LIN {X -0.059,Y -676.284,Z 1223.528,A 0.000,B 0.000,C 90.000,E1 131.024} C_DIS
LIN {X 0.179,Y -679.882,Z 1223.520,A 0.000,B 0.000,C 90.000,E1 129.564} C_DIS
LIN {X 0.002,Y -682.891,Z 1223.513,A 0.000,B 0.000,C 90.000,E1 128.382} C_DIS
LIN {X 0.032,Y -686.511,Z 1223.505,A 0.000,B 0.000,C 90.000,E1 126.950} C_DIS
LIN {X -0.093,Y -688.857,Z 1223.500,A 0.000,B 0.000,C 90.000,E1 126.011} C_DIS
LIN {X -0.354,Y -692.133,Z 1223.492,A 0.000,B 0.000,C 90.000,E1 124.612} C_DIS
LIN {X -0.210,Y -694.745,Z 1223.486,A 0.000,B 0.000,C 90.000,E1 123.420} C_DIS
LIN {X 0.177,Y -697.295,Z 1223.479,A 0.000,B 0.000,C 90.000,E1 122.212} C_DIS
LIN {X 0.274,Y -700.099,Z 1223.471,A 0.000,B 0.000,C 90.000,E1 120.797} C_DIS
LIN {X 0.130,Y -701.847,Z 1223.466,A 0.000,B 0.000,C 90.000,E1 119.873} C_DIS
LIN {X 0.287,Y -703.893,Z 1223.460,A 0.000,B 0.000,C 90.000,E1 118.693} C_DIS
LIN {X -0.100,Y -704.903,Z 1223.456,A 0.000,B 0.000,C 90.000,E1 118.025} C_DIS
LIN {X -0.188,Y -705.601,Z 1223.452,A 0.000,B 0.000,C 90.000,E1 117.334} C_DIS
LIN {X 0.351,Y -706.241,Z 1223.447,A 0.000,B 0.000,C 90.000,E1 116.360} C_DIS
LIN {X -0.348,Y -706.468,Z 1223.443,A 0.000,B 0.000,C 90.000,E1 115.720} C_DIS
LIN {X -0.408,Y -706.297,Z 1223.439,A 0.000,B 0.000,C 90.000,E1 115.027} C_DIS
LIN {X 0.176,Y -705.957,Z 1223.436,A 0.000,B 0.000,C 90.000,E1 114.515} C_DIS
LIN {X -0.177,Y -705.023,Z 1223.434,A 0.000,B 0.000,C 90.000,E1 114.079} C_DIS
LIN {X 0.110,Y -704.351,Z 1223.432,A 0.000,B 0.000,C 90.000,E1 113.823} C_DIS
LIN {X -0.251,Y -702.302,Z 1223.430,A 0.000,B 0.000,C 90.000,E1 113.387} C_DIS
LIN {X -0.112,Y -701.601,Z 1223.429,A 0.000,B 0.000,C 90.000,E1 113.259} C_DIS
LIN {X 0.025,Y -700.554,Z 1223.429,A 0.000,B 0.000,C 90.000,E1 113.131} C_DIS
LIN {X -0.062,Y -695.166,Z 1223.426,A 0.000,B 0.000,C 90.000,E1 112.695} C_DIS
LIN {X -0.096,Y -693.311,Z 1223.426,A 0.000,B 0.000,C 90.000,E1 112.589} C_DIS
LIN {X 0.260,Y -686.621,Z 1223.424,A 0.000,B 0.000,C 90.000,E1 112.333} C_DIS
LIN {X -0.232,Y -684.453,Z 1223.424,A 0.000,B 0.000,C 90.000,E1 112.333} C_DIS
LIN {X -0.007,Y -677.105,Z 1223.424,A 0.000,B 0.000,C 90.000,E1 112.280} C_DIS
LIN {X -0.061,Y -614.428,Z 1223.424,A 0.000,B 0.000,C 90.000,E1 112.280} C_DIS
LIN {X 0.085,Y -612.192,Z 1223.423,A 0.000,B 0.000,C 90.000,E1 112.153} C_DIS
LIN {X -0.235,Y -608.439,Z 1223.422,A 0.000,B 0.000,C 90.000,E1 111.897} C_DIS
LIN {X -0.060,Y -607.204,Z 1223.421,A 0.000,B 0.000,C 90.000,E1 111.770} C_DIS
LIN {X 0.199,Y -605.431,Z 1223.420,A 0.000,B 0.000,C 90.000,E1 111.535} C_DIS
LIN {X 0.044,Y -604.843,Z 1223.419,A 0.000,B 0.000,C 90.000,E1 111.354} C_DIS
LIN {X 0.323,Y -605.149,Z 1223.417,A 0.000,B 0.000,C 90.000,E1 111.099} C_DIS
LIN {X 0.288,Y -605.464,Z 1223.417,A 0.000,B 0.000,C 90.000,E1 110.972} C_DIS
LIN {X -0.099,Y -607.826,Z 1223.413,A 0.000,B 0.000,C 90.000,E1 110.355} C_DIS
LIN {X -0.270,Y -608.959,Z 1223.412,A 0.000,B 0.000,C 90.000,E1 110.120} C_DIS
LIN {X -0.091,Y -612.081,Z 1223.407,A 0.000,B 0.000,C 90.000,E1 109.322} C_DIS
LIN {X 0.203,Y -616.524,Z 1223.400,A 0.000,B 0.000,C 90.000,E1 108.000} C_DIS
LIN {X -0.038,Y -617.374,Z 1223.399,A 0.000,B 0.000,C 90.000,E1 107.764} C_DIS
LIN {X 0.266,Y -619.489,Z 1223.396,A 0.000,B 0.000,C 90.000,E1 107.221} C_DIS
LIN {X -0.074,Y -624.283,Z 1223.389,A 0.000,B 0.000,C 90.000,E1 105.969} C_DIS
LIN {X 0.274,Y -626.084,Z 1223.386,A 0.000,B 0.000,C 90.000,E1 105.426} C_DIS
LIN {X -0.339,Y -628.318,Z 1223.382,A 0.000,B 0.000,C 90.000,E1 104.717} C_DIS
LIN {X -0.168,Y -630.033,Z 1223.377,A 0.000,B 0.000,C 90.000,E1 103.939} C_DIS
LIN {X 0.057,Y -630.911,Z 1223.375,A 0.000,B 0.000,C 90.000,E1 103.411} C_DIS
LIN {X 0.290,Y -631.567,Z 1223.372,A 0.000,B 0.000,C 90.000,E1 102.883} C_DIS
LIN {X 0.339,Y -631.709,Z 1223.368,A 0.000,B 0.000,C 90.000,E1 102.119} C_DIS
LIN {X -0.167,Y -631.385,Z 1223.365,A 0.000,B 0.000,C 90.000,E1 101.658} C_DIS
LIN {X 0.072,Y -630.629,Z 1223.362,A 0.000,B 0.000,C 90.000,E1 101.130} C_DIS
LIN {X 0.108,Y -628.943,Z 1223.358,A 0.000,B 0.000,C 90.000,E1 100.366} C_DIS
LIN {X -0.202,Y -628.261,Z 1223.356,A 0.000,B 0.000,C 90.000,E1 100.141} C_DIS
LIN {X 0.216,Y -627.442,Z 1223.355,A 0.000,B 0.000,C 90.000,E1 99.849} C_DIS
LIN {X -0.195,Y -625.511,Z 1223.352,A 0.000,B 0.000,C 90.000,E1 99.378} C_DIS
LIN {X -0.104,Y -623.269,Z 1223.349,A 0.000,B 0.000,C 90.000,E1 98.859} C_DIS
LIN {X -0.026,Y -620.545,Z 1223.346,A 0.000,B 0.000,C 90.000,E1 98.341} C_DIS
LIN {X -0.256,Y -618.750,Z 1223.345,A 0.000,B 0.000,C 90.000,E1 98.106} C_DIS
LIN {X -0.207,Y -614.791,Z 1223.342,A 0.000,B 0.000,C 90.000,E1 97.587} C_DIS
LIN {X -0.016,Y -611.544,Z 1223.340,A 0.000,B 0.000,C 90.000,E1 97.182} C_DIS
LIN {X 0.019,Y -606.606,Z 1223.337,A 0.000,B 0.000,C 90.000,E1 96.663} C_DIS
LIN {X -0.266,Y -602.361,Z 1223.335,A 0.000,B 0.000,C 90.000,E1 96.315} C_DIS
LIN {X 0.299,Y -598.150,Z 1223.333,A 0.000,B 0.000,C 90.000,E1 95.910} C_DIS
LIN {X -0.153,Y -592.184,Z 1223.331,A 0.000,B 0.000,C 90.000,E1 95.511} C_DIS
LIN {X 0.039,Y -584.245,Z 1223.328,A 0.000,B 0.000,C 90.000,E1 94.992} C_DIS
LIN {X -0.114,Y -577.272,Z 1223.326,A 0.000,B 0.000,C 90.000,E1 94.645} C_DIS
LIN {X 0.264,Y -572.044,Z 1223.324,A 0.000,B 0.000,C 90.000,E1 94.359} C_DIS
LIN {X -0.023,Y -566.787,Z 1223.323,A 0.000,B 0.000,C 90.000,E1 94.073} C_DIS
LIN {X -0.250,Y -564.966,Z 1223.320,A 0.000,B 0.000,C 90.000,E1 93.669} C_DIS
LIN {X -0.066,Y -564.757,Z 1223.320,A 0.000,B 0.000,C 90.000,E1 93.612} C_DIS
LIN {X -0.108,Y -564.741,Z 1223.320,A 0.000,B 0.000,C 90.000,E1 93.612} C_DIS
LIN {X 0.082,Y -564.561,Z 1223.318,A 0.000,B 0.000,C 90.000,E1 93.154} C_DIS
LIN {X -0.022,Y -564.983,Z 1223.312,A 0.000,B 0.000,C 90.000,E1 92.064} C_DIS
LIN {X 0.216,Y -566.310,Z 1223.301,A 0.000,B 0.000,C 90.000,E1 90.115} C_DIS
LIN {X -0.215,Y -567.482,Z 1223.292,A 0.000,B 0.000,C 90.000,E1 88.511} C_DIS
LIN {X 0.105,Y -568.886,Z 1223.281,A 0.000,B 0.000,C 90.000,E1 86.560} C_DIS
LIN {X -0.225,Y -570.213,Z 1223.272,A 0.000,B 0.000,C 90.000,E1 84.951} C_DIS
LIN {X -0.091,Y -571.449,Z 1223.264,A 0.000,B 0.000,C 90.000,E1 83.571} C_DIS
LIN {X 0.124,Y -572.711,Z 1223.257,A 0.000,B 0.000,C 90.000,E1 82.186} C_DIS
LIN {X 0.079,Y -574.094,Z 1223.248,A 0.000,B 0.000,C 90.000,E1 80.557} C_DIS
LIN {X 0.227,Y -574.850,Z 1223.242,A 0.000,B 0.000,C 90.000,E1 79.454} C_DIS
LIN {X 0.223,Y -575.919,Z 1223.233,A 0.000,B 0.000,C 90.000,E1 77.825} C_DIS
LIN {X 0.273,Y -576.748,Z 1223.225,A 0.000,B 0.000,C 90.000,E1 76.464} C_DIS
LIN {X 0.001,Y -577.635,Z 1223.216,A 0.000,B 0.000,C 90.000,E1 74.866} C_DIS
LIN {X -0.262,Y -578.504,Z 1223.207,A 0.000,B 0.000,C 90.000,E1 73.268} C_DIS
LIN {X -0.178,Y -579.420,Z 1223.198,A 0.000,B 0.000,C 90.000,E1 71.638} C_DIS
LIN {X 0.281,Y -580.252,Z 1223.190,A 0.000,B 0.000,C 90.000,E1 70.242} C_DIS
LIN {X -0.044,Y -581.854,Z 1223.177,A 0.000,B 0.000,C 90.000,E1 67.847} C_DIS
LIN {X 0.121,Y -583.018,Z 1223.169,A 0.000,B 0.000,C 90.000,E1 66.485} C_DIS
LIN {X 0.007,Y -584.278,Z 1223.162,A 0.000,B 0.000,C 90.000,E1 65.153} C_DIS
LIN {X 0.205,Y -585.938,Z 1223.152,A 0.000,B 0.000,C 90.000,E1 63.256} C_DIS
LIN {X 0.173,Y -587.852,Z 1223.141,A 0.000,B 0.000,C 90.000,E1 61.385} C_DIS
LIN {X -0.115,Y -589.238,Z 1223.134,A 0.000,B 0.000,C 90.000,E1 60.078} C_DIS
LIN {X -0.087,Y -590.605,Z 1223.126,A 0.000,B 0.000,C 90.000,E1 58.742} C_DIS
LIN {X 0.281,Y -591.835,Z 1223.119,A 0.000,B 0.000,C 90.000,E1 57.375} C_DIS
LIN {X -0.149,Y -592.950,Z 1223.112,A 0.000,B 0.000,C 90.000,E1 56.087} C_DIS
LIN {X -0.235,Y -594.028,Z 1223.104,A 0.000,B 0.000,C 90.000,E1 54.769} C_DIS
LIN {X 0.043,Y -595.053,Z 1223.097,A 0.000,B 0.000,C 90.000,E1 53.417} C_DIS
LIN {X -0.134,Y -596.040,Z 1223.089,A 0.000,B 0.000,C 90.000,E1 52.110} C_DIS
LIN {X -0.295,Y -597.046,Z 1223.082,A 0.000,B 0.000,C 90.000,E1 50.803} C_DIS
LIN {X -0.065,Y -597.586,Z 1223.075,A 0.000,B 0.000,C 90.000,E1 49.461} C_DIS
LIN {X -0.281,Y -598.222,Z 1223.068,A 0.000,B 0.000,C 90.000,E1 48.162} C_DIS
LIN {X 0.352,Y -598.496,Z 1223.063,A 0.000,B 0.000,C 90.000,E1 47.310} C_DIS
LIN {X -0.076,Y -598.805,Z 1223.057,A 0.000,B 0.000,C 90.000,E1 46.296} C_DIS
LIN {X -0.085,Y -598.864,Z 1223.051,A 0.000,B 0.000,C 90.000,E1 45.243} C_DIS
LIN {X -0.092,Y -598.785,Z 1223.046,A 0.000,B 0.000,C 90.000,E1 44.190} C_DIS
LIN {X 0.109,Y -598.584,Z 1223.041,A 0.000,B 0.000,C 90.000,E1 43.380} C_DIS
LIN {X 0.122,Y -598.073,Z 1223.035,A 0.000,B 0.000,C 90.000,E1 42.324} C_DIS
LIN {X 0.310,Y -597.379,Z 1223.028,A 0.000,B 0.000,C 90.000,E1 40.987} C_DIS
LIN {X -0.301,Y -596.610,Z 1223.021,A 0.000,B 0.000,C 90.000,E1 39.725} C_DIS
LIN {X -0.086,Y -595.582,Z 1223.013,A 0.000,B 0.000,C 90.000,E1 38.382} C_DIS
LIN {X -0.015,Y -594.501,Z 1223.007,A 0.000,B 0.000,C 90.000,E1 37.317} C_DIS
LIN {X 0.048,Y -593.129,Z 1223.001,A 0.000,B 0.000,C 90.000,E1 36.251} C_DIS
LIN {X 0.091,Y -591.547,Z 1222.996,A 0.000,B 0.000,C 90.000,E1 35.185} C_DIS
LIN {X -0.100,Y -590.059,Z 1222.991,A 0.000,B 0.000,C 90.000,E1 34.405} C_DIS
LIN {X 0.177,Y -588.396,Z 1222.987,A 0.000,B 0.000,C 90.000,E1 33.579} C_DIS
LIN {X -0.247,Y -587.057,Z 1222.984,A 0.000,B 0.000,C 90.000,E1 33.086} C_DIS
LIN {X -0.138,Y -584.159,Z 1222.978,A 0.000,B 0.000,C 90.000,E1 32.005} C_DIS
LIN {X -0.098,Y -582.461,Z 1222.975,A 0.000,B 0.000,C 90.000,E1 31.465} C_DIS
LIN {X -0.071,Y -580.560,Z 1222.972,A 0.000,B 0.000,C 90.000,E1 30.924} C_DIS
LIN {X -0.204,Y -577.327,Z 1222.967,A 0.000,B 0.000,C 90.000,E1 30.129} C_DIS
LIN {X 0.284,Y -574.974,Z 1222.964,A 0.000,B 0.000,C 90.000,E1 29.539} C_DIS
LIN {X -0.027,Y -572.455,Z 1222.961,A 0.000,B 0.000,C 90.000,E1 29.027} C_DIS
LIN {X -0.164,Y -568.879,Z 1222.958,A 0.000,B 0.000,C 90.000,E1 28.359} C_DIS
LIN {X 0.072,Y -564.280,Z 1222.953,A 0.000,B 0.000,C 90.000,E1 27.513} C_DIS
LIN {X 0.099,Y -560.113,Z 1222.949,A 0.000,B 0.000,C 90.000,E1 26.821} C_DIS
LIN {X -0.161,Y -555.569,Z 1222.945,A 0.000,B 0.000,C 90.000,E1 26.155} C_DIS
LIN {X -0.095,Y -551.637,Z 1222.942,A 0.000,B 0.000,C 90.000,E1 25.591} C_DIS
LIN {X 0.063,Y -548.547,Z 1222.940,A 0.000,B 0.000,C 90.000,E1 25.155} C_DIS
LIN {X -0.168,Y -541.798,Z 1222.935,A 0.000,B 0.000,C 90.000,E1 24.335} C_DIS
LIN {X 0.024,Y -534.509,Z 1222.930,A 0.000,B 0.000,C 90.000,E1 23.462} C_DIS
LIN {X -0.138,Y -526.938,Z 1222.926,A 0.000,B 0.000,C 90.000,E1 22.642} C_DIS
LIN {X -0.090,Y -521.762,Z 1222.923,A 0.000,B 0.000,C 90.000,E1 22.078} C_DIS
LIN {X -0.152,Y -510.874,Z 1222.917,A 0.000,B 0.000,C 90.000,E1 20.972} C_DIS
LIN {X -0.057,Y -499.892,Z 1222.911,A 0.000,B 0.000,C 90.000,E1 19.885} C_DIS
LIN {X -0.074,Y -489.981,Z 1222.905,A 0.000,B 0.000,C 90.000,E1 18.960} C_DIS
LIN {X -0.159,Y -482.654,Z 1222.902,A 0.000,B 0.000,C 90.000,E1 18.308} C_DIS
LIN {X -0.043,Y -471.100,Z 1222.896,A 0.000,B 0.000,C 90.000,E1 17.275} C_DIS
LIN {X 0.101,Y -457.930,Z 1222.889,A 0.000,B 0.000,C 90.000,E1 16.079} C_DIS
LIN {X -0.247,Y -440.285,Z 1222.880,A 0.000,B 0.000,C 90.000,E1 14.481} C_DIS
LIN {X -0.047,Y -420.268,Z 1222.869,A 0.000,B 0.000,C 90.000,E1 12.411} C_DIS
LIN {X 0.106,Y -403.560,Z 1222.858,A 0.000,B 0.000,C 90.000,E1 10.489} C_DIS
LIN {X -0.208,Y -398.266,Z 1222.855,A 0.000,B 0.000,C 90.000,E1 9.849} C_DIS
LIN {X 0.192,Y -394.919,Z 1222.852,A 0.000,B 0.000,C 90.000,E1 9.265} C_DIS
LIN {X 0.114,Y -393.810,Z 1222.850,A 0.000,B 0.000,C 90.000,E1 8.973} C_DIS
LIN {X 0.076,Y -393.799,Z 1222.850,A 0.000,B 0.000,C 90.000,E1 8.973} C_DIS
LIN {X 0.084,Y -394.025,Z 1222.848,A 0.000,B 0.000,C 90.000,E1 8.690} C_DIS
LIN {X 0.105,Y -394.035,Z 1222.848,A 0.000,B 0.000,C 90.000,E1 8.681} C_DIS
LIN {X 0.042,Y -396.943,Z 1222.845,A 0.000,B 0.000,C 90.000,E1 8.049} C_DIS
LIN {X 0.063,Y -399.821,Z 1222.843,A 0.000,B 0.000,C 90.000,E1 7.701} C_DIS
LIN {X 0.073,Y -401.418,Z 1222.842,A 0.000,B 0.000,C 90.000,E1 7.530} C_DIS
LIN {X -0.127,Y -405.153,Z 1222.840,A 0.000,B 0.000,C 90.000,E1 7.239} C_DIS
LIN {X -0.195,Y -418.242,Z 1222.835,A 0.000,B 0.000,C 90.000,E1 6.258} C_DIS
LIN {X -0.178,Y -432.604,Z 1222.829,A 0.000,B 0.000,C 90.000,E1 5.163} C_DIS
LIN {X -0.107,Y -443.683,Z 1222.824,A 0.000,B 0.000,C 90.000,E1 4.302} C_DIS
LIN {X -0.046,Y -456.342,Z 1222.818,A 0.000,B 0.000,C 90.000,E1 3.326} C_DIS
LIN {X 0.101,Y -465.722,Z 1222.814,A 0.000,B 0.000,C 90.000,E1 2.579} C_DIS
LIN {X -0.192,Y -471.854,Z 1222.812,A 0.000,B 0.000,C 90.000,E1 2.121} C_DIS
LIN {X 0.171,Y -479.159,Z 1222.808,A 0.000,B 0.000,C 90.000,E1 1.432} C_DIS
LIN {X 0.000,Y -484.954,Z 1222.805,A 0.000,B 0.000,C 90.000,E1 0.917} C_DIS
LIN {X 0.212,Y -491.536,Z 1222.802,A 0.000,B 0.000,C 90.000,E1 0.229} C_DIS
LIN {X 0.170,Y -498.380,Z 1222.797,A 0.000,B 0.000,C 90.000,E1 359.484} C_DIS
LIN {X 0.158,Y -504.685,Z 1222.793,A 0.000,B 0.000,C 90.000,E1 358.740} C_DIS
LIN {X 0.201,Y -510.430,Z 1222.789,A 0.000,B 0.000,C 90.000,E1 357.993} C_DIS
LIN {X 0.243,Y -515.707,Z 1222.785,A 0.000,B 0.000,C 90.000,E1 357.249} C_DIS
LIN {X -0.163,Y -520.650,Z 1222.781,A 0.000,B 0.000,C 90.000,E1 356.560} C_DIS
LIN {X -0.277,Y -524.346,Z 1222.778,A 0.000,B 0.000,C 90.000,E1 355.988} C_DIS
LIN {X -0.087,Y -528.528,Z 1222.774,A 0.000,B 0.000,C 90.000,E1 355.241} C_DIS
LIN {X -0.108,Y -531.614,Z 1222.770,A 0.000,B 0.000,C 90.000,E1 354.666} C_DIS
LIN {X -0.068,Y -535.706,Z 1222.766,A 0.000,B 0.000,C 90.000,E1 353.799} C_DIS
LIN {X 0.239,Y -537.669,Z 1222.763,A 0.000,B 0.000,C 90.000,E1 353.337} C_DIS
LIN {X -0.185,Y -541.159,Z 1222.758,A 0.000,B 0.000,C 90.000,E1 352.527} C_DIS
LIN {X -0.117,Y -543.342,Z 1222.755,A 0.000,B 0.000,C 90.000,E1 351.951} C_DIS
LIN {X 0.050,Y -546.331,Z 1222.750,A 0.000,B 0.000,C 90.000,E1 351.084} C_DIS
LIN {X -0.296,Y -549.011,Z 1222.746,A 0.000,B 0.000,C 90.000,E1 350.274} C_DIS
LIN {X 0.251,Y -552.968,Z 1222.738,A 0.000,B 0.000,C 90.000,E1 348.814} C_DIS
LIN {X 0.202,Y -555.871,Z 1222.732,A 0.000,B 0.000,C 90.000,E1 347.701} C_DIS
LIN {X 0.056,Y -557.799,Z 1222.727,A 0.000,B 0.000,C 90.000,E1 346.881} C_DIS
LIN {X -0.197,Y -560.745,Z 1222.719,A 0.000,B 0.000,C 90.000,E1 345.519} C_DIS
LIN {X -0.005,Y -562.954,Z 1222.713,A 0.000,B 0.000,C 90.000,E1 344.393} C_DIS
LIN {X 0.212,Y -564.938,Z 1222.707,A 0.000,B 0.000,C 90.000,E1 343.268} C_DIS
LIN {X 0.078,Y -566.653,Z 1222.701,A 0.000,B 0.000,C 90.000,E1 342.181} C_DIS
LIN {X 0.309,Y -568.505,Z 1222.693,A 0.000,B 0.000,C 90.000,E1 340.786} C_DIS
LIN {X -0.119,Y -569.478,Z 1222.689,A 0.000,B 0.000,C 90.000,E1 340.007} C_DIS
LIN {X 0.186,Y -570.159,Z 1222.684,A 0.000,B 0.000,C 90.000,E1 339.156} C_DIS
LIN {X 0.175,Y -570.625,Z 1222.680,A 0.000,B 0.000,C 90.000,E1 338.337} C_DIS
LIN {X -0.038,Y -570.854,Z 1222.675,A 0.000,B 0.000,C 90.000,E1 337.539} C_DIS
LIN {X 0.097,Y -570.545,Z 1222.669,A 0.000,B 0.000,C 90.000,E1 336.433} C_DIS
LIN {X -0.247,Y -570.248,Z 1222.666,A 0.000,B 0.000,C 90.000,E1 335.921} C_DIS
LIN {X -0.242,Y -569.376,Z 1222.662,A 0.000,B 0.000,C 90.000,E1 335.101} C_DIS
LIN {X -0.246,Y -568.326,Z 1222.657,A 0.000,B 0.000,C 90.000,E1 334.280} C_DIS
LIN {X -0.013,Y -566.722,Z 1222.652,A 0.000,B 0.000,C 90.000,E1 333.435} C_DIS
LIN {X -0.049,Y -564.801,Z 1222.648,A 0.000,B 0.000,C 90.000,E1 332.615} C_DIS
LIN {X 0.340,Y -563.446,Z 1222.645,A 0.000,B 0.000,C 90.000,E1 332.025} C_DIS
LIN {X -0.042,Y -561.824,Z 1222.642,A 0.000,B 0.000,C 90.000,E1 331.513} C_DIS
LIN {X -0.238,Y -560.916,Z 1222.640,A 0.000,B 0.000,C 90.000,E1 331.257} C_DIS
LIN {X 0.123,Y -558.717,Z 1222.637,A 0.000,B 0.000,C 90.000,E1 330.667} C_DIS
LIN {X -0.234,Y -554.940,Z 1222.633,A 0.000,B 0.000,C 90.000,E1 329.871} C_DIS
LIN {X 0.126,Y -550.429,Z 1222.628,A 0.000,B 0.000,C 90.000,E1 328.997} C_DIS
LIN {X -0.193,Y -546.066,Z 1222.624,A 0.000,B 0.000,C 90.000,E1 328.329} C_DIS
LIN {X 0.200,Y -541.331,Z 1222.620,A 0.000,B 0.000,C 90.000,E1 327.582} C_DIS
LIN {X 0.082,Y -538.220,Z 1222.618,A 0.000,B 0.000,C 90.000,E1 327.168} C_DIS
LIN {X 0.233,Y -529.278,Z 1222.611,A 0.000,B 0.000,C 90.000,E1 326.008} C_DIS
LIN {X -0.133,Y -517.890,Z 1222.603,A 0.000,B 0.000,C 90.000,E1 324.609} C_DIS
LIN {X -0.023,Y -514.390,Z 1222.600,A 0.000,B 0.000,C 90.000,E1 324.069} C_DIS
LIN {X 0.074,Y -511.531,Z 1222.598,A 0.000,B 0.000,C 90.000,E1 323.543} C_DIS
LIN {X -0.008,Y -509.878,Z 1222.595,A 0.000,B 0.000,C 90.000,E1 323.084} C_DIS
LIN {X 0.103,Y -509.411,Z 1222.594,A 0.000,B 0.000,C 90.000,E1 322.924} C_DIS
LIN {X 0.088,Y -508.395,Z 1222.591,A 0.000,B 0.000,C 90.000,E1 322.396} C_DIS
LIN {X -0.004,Y -508.026,Z 1222.590,A 0.000,B 0.000,C 90.000,E1 322.110} C_DIS
LIN {X -0.159,Y -507.568,Z 1222.585,A 0.000,B 0.000,C 90.000,E1 321.251} C_DIS
LIN {X -0.036,Y -507.499,Z 1222.581,A 0.000,B 0.000,C 90.000,E1 320.642} C_DIS
LIN {X 0.049,Y -509.039,Z 1222.567,A 0.000,B 0.000,C 90.000,E1 317.957} C_DIS
LIN {X 0.188,Y -509.856,Z 1222.558,A 0.000,B 0.000,C 90.000,E1 316.458} C_DIS
LIN {X -0.021,Y -510.592,Z 1222.550,A 0.000,B 0.000,C 90.000,E1 315.000} C_DIS
LIN {X -0.066,Y -511.503,Z 1222.539,A 0.000,B 0.000,C 90.000,E1 312.933} C_DIS
LIN {X -0.057,Y -512.465,Z 1222.527,A 0.000,B 0.000,C 90.000,E1 310.862} C_DIS
LIN {X 0.193,Y -513.080,Z 1222.519,A 0.000,B 0.000,C 90.000,E1 309.358} C_DIS
LIN {X 0.280,Y -513.374,Z 1222.514,A 0.000,B 0.000,C 90.000,E1 308.463} C_DIS
LIN {X -0.015,Y -514.155,Z 1222.501,A 0.000,B 0.000,C 90.000,E1 306.137} C_DIS
LIN {X 0.087,Y -514.783,Z 1222.491,A 0.000,B 0.000,C 90.000,E1 304.358} C_DIS
LIN {X 0.144,Y -515.305,Z 1222.483,A 0.000,B 0.000,C 90.000,E1 302.880} C_DIS
LIN {X 0.081,Y -515.612,Z 1222.475,A 0.000,B 0.000,C 90.000,E1 301.416} C_DIS
LIN {X 0.033,Y -515.841,Z 1222.466,A 0.000,B 0.000,C 90.000,E1 299.951} C_DIS
LIN {X 0.075,Y -515.978,Z 1222.460,A 0.000,B 0.000,C 90.000,E1 298.771} C_DIS
LIN {X 0.015,Y -516.132,Z 1222.452,A 0.000,B 0.000,C 90.000,E1 297.308} C_DIS
LIN {X 0.060,Y -516.164,Z 1222.442,A 0.000,B 0.000,C 90.000,E1 295.540} C_DIS
LIN {X 0.117,Y -516.315,Z 1222.432,A 0.000,B 0.000,C 90.000,E1 293.770} C_DIS
LIN {X -0.169,Y -516.334,Z 1222.424,A 0.000,B 0.000,C 90.000,E1 292.333} C_DIS
LIN {X 0.011,Y -516.013,Z 1222.416,A 0.000,B 0.000,C 90.000,E1 290.844} C_DIS
LIN {X -0.133,Y -515.448,Z 1222.409,A 0.000,B 0.000,C 90.000,E1 289.685} C_DIS
LIN {X 0.280,Y -514.640,Z 1222.400,A 0.000,B 0.000,C 90.000,E1 287.873} C_DIS
LIN {X -0.083,Y -513.936,Z 1222.391,A 0.000,B 0.000,C 90.000,E1 286.441} C_DIS
LIN {X 0.039,Y -513.160,Z 1222.383,A 0.000,B 0.000,C 90.000,E1 284.954} C_DIS
LIN {X 0.075,Y -511.927,Z 1222.372,A 0.000,B 0.000,C 90.000,E1 282.883} C_DIS
LIN {X -0.082,Y -510.903,Z 1222.363,A 0.000,B 0.000,C 90.000,E1 281.422} C_DIS
LIN {X -0.183,Y -510.261,Z 1222.359,A 0.000,B 0.000,C 90.000,E1 280.546} C_DIS
LIN {X 0.005,Y -509.071,Z 1222.349,A 0.000,B 0.000,C 90.000,E1 278.746} C_DIS
LIN {X -0.008,Y -507.495,Z 1222.335,A 0.000,B 0.000,C 90.000,E1 276.372} C_DIS
LIN {X -0.194,Y -506.211,Z 1222.322,A 0.000,B 0.000,C 90.000,E1 274.012} C_DIS
LIN {X 0.020,Y -505.717,Z 1222.317,A 0.000,B 0.000,C 90.000,E1 273.094} C_DIS
LIN {X 0.010,Y -504.723,Z 1222.309,A 0.000,B 0.000,C 90.000,E1 271.604} C_DIS
LIN {X -0.024,Y -503.741,Z 1222.301,A 0.000,B 0.000,C 90.000,E1 270.115} C_DIS
LIN {X -0.076,Y -502.931,Z 1222.292,A 0.000,B 0.000,C 90.000,E1 268.625} C_DIS
LIN {X 0.155,Y -501.732,Z 1222.281,A 0.000,B 0.000,C 90.000,E1 266.502} C_DIS
LIN {X 0.194,Y -500.946,Z 1222.274,A 0.000,B 0.000,C 90.000,E1 265.298} C_DIS
LIN {X 0.175,Y -499.866,Z 1222.266,A 0.000,B 0.000,C 90.000,E1 263.799} C_DIS
LIN {X 0.222,Y -498.842,Z 1222.259,A 0.000,B 0.000,C 90.000,E1 262.591} C_DIS
LIN {X 0.060,Y -496.881,Z 1222.247,A 0.000,B 0.000,C 90.000,E1 260.500} C_DIS
LIN {X 0.030,Y -495.589,Z 1222.239,A 0.000,B 0.000,C 90.000,E1 258.993} C_DIS
LIN {X -0.105,Y -493.443,Z 1222.224,A 0.000,B 0.000,C 90.000,E1 256.284} C_DIS
LIN {X -0.010,Y -492.418,Z 1222.215,A 0.000,B 0.000,C 90.000,E1 254.755} C_DIS
LIN {X 0.173,Y -490.733,Z 1222.198,A 0.000,B 0.000,C 90.000,E1 251.692} C_DIS
LIN {X 0.036,Y -489.858,Z 1222.188,A 0.000,B 0.000,C 90.000,E1 249.880} C_DIS
LIN {X 0.156,Y -489.217,Z 1222.182,A 0.000,B 0.000,C 90.000,E1 248.646} C_DIS
LIN {X 0.269,Y -488.456,Z 1222.175,A 0.000,B 0.000,C 90.000,E1 247.411} C_DIS
LIN {X -0.081,Y -487.566,Z 1222.168,A 0.000,B 0.000,C 90.000,E1 246.230} C_DIS
LIN {X -0.218,Y -485.933,Z 1222.158,A 0.000,B 0.000,C 90.000,E1 244.409} C_DIS
LIN {X -0.191,Y -484.416,Z 1222.149,A 0.000,B 0.000,C 90.000,E1 242.871} C_DIS
LIN {X 0.246,Y -483.543,Z 1222.144,A 0.000,B 0.000,C 90.000,E1 241.897} C_DIS
LIN {X -0.188,Y -482.164,Z 1222.137,A 0.000,B 0.000,C 90.000,E1 240.717} C_DIS
LIN {X -0.197,Y -481.087,Z 1222.132,A 0.000,B 0.000,C 90.000,E1 239.793} C_DIS
LIN {X 0.195,Y -479.355,Z 1222.124,A 0.000,B 0.000,C 90.000,E1 238.201} C_DIS
LIN {X -0.073,Y -477.160,Z 1222.113,A 0.000,B 0.000,C 90.000,E1 236.373} C_DIS
LIN {X 0.106,Y -474.360,Z 1222.099,A 0.000,B 0.000,C 90.000,E1 233.863} C_DIS
LIN {X -0.006,Y -472.691,Z 1222.091,A 0.000,B 0.000,C 90.000,E1 232.316} C_DIS
LIN {X -0.139,Y -470.311,Z 1222.077,A 0.000,B 0.000,C 90.000,E1 229.828} C_DIS
LIN {X -0.016,Y -468.939,Z 1222.068,A 0.000,B 0.000,C 90.000,E1 228.243} C_DIS
LIN {X -0.130,Y -466.942,Z 1222.056,A 0.000,B 0.000,C 90.000,E1 226.053} C_DIS
LIN {X -0.138,Y -465.036,Z 1222.000,A 0.000,B 0.000,C 90.000,E1 215.931} C_DIS
LIN {X 0.059,Y -467.545,Z 1221.977,A 0.000,B 0.000,C 90.000,E1 211.799} C_DIS
LIN {X 0.198,Y -469.058,Z 1221.968,A 0.000,B 0.000,C 90.000,E1 210.207} C_DIS
LIN {X 0.169,Y -472.175,Z 1221.952,A 0.000,B 0.000,C 90.000,E1 207.385} C_DIS
LIN {X 0.050,Y -475.252,Z 1221.938,A 0.000,B 0.000,C 90.000,E1 204.899} C_DIS
LIN {X 0.043,Y -480.522,Z 1221.919,A 0.000,B 0.000,C 90.000,E1 201.482} C_DIS
LIN {X -0.233,Y -487.846,Z 1221.899,A 0.000,B 0.000,C 90.000,E1 197.819} C_DIS
LIN {X 0.130,Y -495.918,Z 1221.880,A 0.000,B 0.000,C 90.000,E1 194.426} C_DIS
LIN {X -0.225,Y -501.638,Z 1221.869,A 0.000,B 0.000,C 90.000,E1 192.355} C_DIS
LIN {X -0.057,Y -505.777,Z 1221.860,A 0.000,B 0.000,C 90.000,E1 190.838} C_DIS
LIN {X 0.029,Y -511.799,Z 1221.849,A 0.000,B 0.000,C 90.000,E1 188.746} C_DIS
LIN {X -0.203,Y -516.239,Z 1221.840,A 0.000,B 0.000,C 90.000,E1 187.296} C_DIS
LIN {X 0.106,Y -519.715,Z 1221.834,A 0.000,B 0.000,C 90.000,E1 186.087} C_DIS
LIN {X -0.160,Y -526.470,Z 1221.821,A 0.000,B 0.000,C 90.000,E1 183.784} C_DIS
LIN {X 0.246,Y -530.750,Z 1221.813,A 0.000,B 0.000,C 90.000,E1 182.293} C_DIS
LIN {X 0.203,Y -534.977,Z 1221.805,A 0.000,B 0.000,C 90.000,E1 180.859} C_DIS
LIN {X 0.226,Y -539.171,Z 1221.797,A 0.000,B 0.000,C 90.000,E1 179.427} C_DIS
LIN {X -0.179,Y -544.022,Z 1221.787,A 0.000,B 0.000,C 90.000,E1 177.764} C_DIS
LIN {X 0.018,Y -547.912,Z 1221.780,A 0.000,B 0.000,C 90.000,E1 176.331} C_DIS
LIN {X -0.230,Y -551.648,Z 1221.772,A 0.000,B 0.000,C 90.000,E1 174.951} C_DIS
LIN {X 0.134,Y -555.249,Z 1221.764,A 0.000,B 0.000,C 90.000,E1 173.514} C_DIS
LIN {X 0.067,Y -558.781,Z 1221.756,A 0.000,B 0.000,C 90.000,E1 172.129} C_DIS
LIN {X -0.005,Y -561.573,Z 1221.750,A 0.000,B 0.000,C 90.000,E1 171.027} C_DIS
LIN {X -0.038,Y -564.376,Z 1221.744,A 0.000,B 0.000,C 90.000,E1 169.926} C_DIS
LIN {X -0.136,Y -568.449,Z 1221.735,A 0.000,B 0.000,C 90.000,E1 168.285} C_DIS
LIN {X -0.142,Y -572.605,Z 1221.726,A 0.000,B 0.000,C 90.000,E1 166.645} C_DIS
LIN {X -0.284,Y -577.657,Z 1221.715,A 0.000,B 0.000,C 90.000,E1 164.755} C_DIS
LIN {X -0.039,Y -586.173,Z 1221.699,A 0.000,B 0.000,C 90.000,E1 161.764} C_DIS
LIN {X 0.065,Y -599.104,Z 1221.678,A 0.000,B 0.000,C 90.000,E1 158.028} C_DIS
LIN {X 0.072,Y -603.122,Z 1221.672,A 0.000,B 0.000,C 90.000,E1 156.975} C_DIS
LIN {X 0.130,Y -607.099,Z 1221.666,A 0.000,B 0.000,C 90.000,E1 155.921} C_DIS
LIN {X -0.363,Y -612.003,Z 1221.659,A 0.000,B 0.000,C 90.000,E1 154.665} C_DIS
LIN {X 0.059,Y -615.769,Z 1221.653,A 0.000,B 0.000,C 90.000,E1 153.589} C_DIS
LIN {X -0.020,Y -619.398,Z 1221.648,A 0.000,B 0.000,C 90.000,E1 152.564} C_DIS
LIN {X 0.239,Y -623.749,Z 1221.641,A 0.000,B 0.000,C 90.000,E1 151.257} C_DIS
LIN {X 0.022,Y -627.175,Z 1221.635,A 0.000,B 0.000,C 90.000,E1 150.255} C_DIS
LIN {X -0.124,Y -631.420,Z 1221.628,A 0.000,B 0.000,C 90.000,E1 148.997} C_DIS
LIN {X 0.158,Y -636.288,Z 1221.619,A 0.000,B 0.000,C 90.000,E1 147.454} C_DIS
LIN {X 0.064,Y -638.577,Z 1221.615,A 0.000,B 0.000,C 90.000,E1 146.707} C_DIS
LIN {X -0.105,Y -642.269,Z 1221.608,A 0.000,B 0.000,C 90.000,E1 145.468} C_DIS
LIN {X -0.330,Y -646.173,Z 1221.600,A 0.000,B 0.000,C 90.000,E1 143.989} C_DIS
LIN {X 0.038,Y -647.958,Z 1221.596,A 0.000,B 0.000,C 90.000,E1 143.210} C_DIS
LIN {X -0.203,Y -651.413,Z 1221.587,A 0.000,B 0.000,C 90.000,E1 141.743} C_DIS
LIN {X -0.318,Y -654.162,Z 1221.581,A 0.000,B 0.000,C 90.000,E1 140.517} C_DIS
LIN {X 0.018,Y -656.881,Z 1221.574,A 0.000,B 0.000,C 90.000,E1 139.256} C_DIS
LIN {X -0.132,Y -660.162,Z 1221.566,A 0.000,B 0.000,C 90.000,E1 137.796} C_DIS
LIN {X 0.222,Y -663.848,Z 1221.556,A 0.000,B 0.000,C 90.000,E1 136.053} C_DIS
LIN {X 0.200,Y -669.057,Z 1221.544,A 0.000,B 0.000,C 90.000,E1 133.866} C_DIS
LIN {X -0.211,Y -672.135,Z 1221.537,A 0.000,B 0.000,C 90.000,E1 132.690} C_DIS
LIN {X -0.052,Y -675.822,Z 1221.529,A 0.000,B 0.000,C 90.000,E1 131.229} C_DIS
LIN {X -0.237,Y -679.972,Z 1221.520,A 0.000,B 0.000,C 90.000,E1 129.564} C_DIS
LIN {X 0.122,Y -682.964,Z 1221.513,A 0.000,B 0.000,C 90.000,E1 128.338} C_DIS
LIN {X -0.384,Y -686.599,Z 1221.505,A 0.000,B 0.000,C 90.000,E1 126.950} C_DIS
LIN {X 0.049,Y -688.934,Z 1221.500,A 0.000,B 0.000,C 90.000,E1 125.964} C_DIS
LIN {X 0.190,Y -692.230,Z 1221.492,A 0.000,B 0.000,C 90.000,E1 124.532} C_DIS
LIN {X -0.398,Y -695.339,Z 1221.484,A 0.000,B 0.000,C 90.000,E1 123.166} C_DIS
LIN {X -0.241,Y -697.365,Z 1221.479,A 0.000,B 0.000,C 90.000,E1 122.212} C_DIS
LIN {X -0.144,Y -700.193,Z 1221.471,A 0.000,B 0.000,C 90.000,E1 120.797} C_DIS
LIN {X -0.352,Y -702.788,Z 1221.463,A 0.000,B 0.000,C 90.000,E1 119.411} C_DIS
LIN {X 0.153,Y -704.332,Z 1221.458,A 0.000,B 0.000,C 90.000,E1 118.437} C_DIS
LIN {X -0.232,Y -705.232,Z 1221.454,A 0.000,B 0.000,C 90.000,E1 117.769} C_DIS
LIN {X 0.007,Y -705.859,Z 1221.450,A 0.000,B 0.000,C 90.000,E1 117.052} C_DIS
LIN {X 0.228,Y -706.403,Z 1221.445,A 0.000,B 0.000,C 90.000,E1 116.104} C_DIS
LIN {X 0.168,Y -706.499,Z 1221.441,A 0.000,B 0.000,C 90.000,E1 115.412} C_DIS
LIN {X 0.115,Y -706.355,Z 1221.439,A 0.000,B 0.000,C 90.000,E1 114.951} C_DIS
LIN {X -0.238,Y -705.958,Z 1221.436,A 0.000,B 0.000,C 90.000,E1 114.515} C_DIS
LIN {X 0.052,Y -705.000,Z 1221.434,A 0.000,B 0.000,C 90.000,E1 114.027} C_DIS
LIN {X -0.303,Y -704.241,Z 1221.432,A 0.000,B 0.000,C 90.000,E1 113.823} C_DIS
LIN {X -0.019,Y -702.197,Z 1221.430,A 0.000,B 0.000,C 90.000,E1 113.334} C_DIS
LIN {X 0.120,Y -701.412,Z 1221.429,A 0.000,B 0.000,C 90.000,E1 113.206} C_DIS
LIN {X 0.258,Y -700.245,Z 1221.428,A 0.000,B 0.000,C 90.000,E1 113.078} C_DIS
LIN {X 0.170,Y -694.653,Z 1221.426,A 0.000,B 0.000,C 90.000,E1 112.642} C_DIS
LIN {X -0.175,Y -692.571,Z 1221.425,A 0.000,B 0.000,C 90.000,E1 112.567} C_DIS
LIN {X 0.023,Y -685.847,Z 1221.424,A 0.000,B 0.000,C 90.000,E1 112.333} C_DIS
LIN {X -0.226,Y -684.511,Z 1221.424,A 0.000,B 0.000,C 90.000,E1 112.333} C_DIS
LIN {X 0.014,Y -676.884,Z 1221.424,A 0.000,B 0.000,C 90.000,E1 112.280} C_DIS
LIN {X -0.020,Y -613.742,Z 1221.424,A 0.000,B 0.000,C 90.000,E1 112.280} C_DIS
LIN {X -0.024,Y -611.226,Z 1221.423,A 0.000,B 0.000,C 90.000,E1 112.153} C_DIS
LIN {X 0.033,Y -607.187,Z 1221.421,A 0.000,B 0.000,C 90.000,E1 111.844} C_DIS
LIN {X -0.061,Y -605.331,Z 1221.420,A 0.000,B 0.000,C 90.000,E1 111.642} C_DIS
LIN {X 0.119,Y -603.890,Z 1221.419,A 0.000,B 0.000,C 90.000,E1 111.482} C_DIS
LIN {X 0.076,Y -603.851,Z 1221.419,A 0.000,B 0.000,C 90.000,E1 111.482} C_DIS
LIN {X 0.308,Y -603.272,Z 1221.418,A 0.000,B 0.000,C 90.000,E1 111.280} C_DIS
LIN {X 0.070,Y -604.117,Z 1221.416,A 0.000,B 0.000,C 90.000,E1 110.844} C_DIS
LIN {X -0.180,Y -605.884,Z 1221.413,A 0.000,B 0.000,C 90.000,E1 110.355} C_DIS
LIN {X -0.239,Y -609.035,Z 1221.409,A 0.000,B 0.000,C 90.000,E1 109.577} C_DIS
LIN {X -0.320,Y -612.624,Z 1221.403,A 0.000,B 0.000,C 90.000,E1 108.544} C_DIS
LIN {X -0.299,Y -615.175,Z 1221.399,A 0.000,B 0.000,C 90.000,E1 107.764} C_DIS
LIN {X -0.011,Y -617.121,Z 1221.396,A 0.000,B 0.000,C 90.000,E1 107.221} C_DIS
LIN {X -0.170,Y -620.941,Z 1221.390,A 0.000,B 0.000,C 90.000,E1 106.205} C_DIS
LIN {X -0.064,Y -623.478,Z 1221.386,A 0.000,B 0.000,C 90.000,E1 105.426} C_DIS
LIN {X -0.097,Y -625.555,Z 1221.381,A 0.000,B 0.000,C 90.000,E1 104.662} C_DIS
LIN {X 0.253,Y -626.750,Z 1221.379,A 0.000,B 0.000,C 90.000,E1 104.120} C_DIS
LIN {X -0.154,Y -627.648,Z 1221.376,A 0.000,B 0.000,C 90.000,E1 103.647} C_DIS
LIN {X 0.056,Y -628.291,Z 1221.373,A 0.000,B 0.000,C 90.000,E1 103.119} C_DIS
LIN {X -0.143,Y -628.508,Z 1221.372,A 0.000,B 0.000,C 90.000,E1 102.883} C_DIS
LIN {X 0.074,Y -628.661,Z 1221.369,A 0.000,B 0.000,C 90.000,E1 102.355} C_DIS
LIN {X 0.292,Y -628.375,Z 1221.366,A 0.000,B 0.000,C 90.000,E1 101.827} C_DIS
LIN {X 0.093,Y -628.085,Z 1221.365,A 0.000,B 0.000,C 90.000,E1 101.591} C_DIS
LIN {X 0.185,Y -627.210,Z 1221.362,A 0.000,B 0.000,C 90.000,E1 101.074} C_DIS
LIN {X -0.221,Y -626.120,Z 1221.359,A 0.000,B 0.000,C 90.000,E1 100.602} C_DIS
LIN {X -0.023,Y -624.646,Z 1221.356,A 0.000,B 0.000,C 90.000,E1 100.074} C_DIS
LIN {X 0.057,Y -622.752,Z 1221.353,A 0.000,B 0.000,C 90.000,E1 99.557} C_DIS
LIN {X 0.067,Y -619.904,Z 1221.350,A 0.000,B 0.000,C 90.000,E1 98.916} C_DIS
LIN {X 0.044,Y -616.126,Z 1221.346,A 0.000,B 0.000,C 90.000,E1 98.276} C_DIS
LIN {X 0.070,Y -612.332,Z 1221.343,A 0.000,B 0.000,C 90.000,E1 97.757} C_DIS
LIN {X -0.102,Y -606.514,Z 1221.340,A 0.000,B 0.000,C 90.000,E1 97.125} C_DIS
LIN {X 0.023,Y -601.218,Z 1221.337,A 0.000,B 0.000,C 90.000,E1 96.606} C_DIS
LIN {X -0.112,Y -595.675,Z 1221.334,A 0.000,B 0.000,C 90.000,E1 96.144} C_DIS
LIN {X 0.104,Y -589.615,Z 1221.332,A 0.000,B 0.000,C 90.000,E1 95.682} C_DIS
LIN {X 0.267,Y -586.410,Z 1221.330,A 0.000,B 0.000,C 90.000,E1 95.454} C_DIS
LIN {X 0.075,Y -578.178,Z 1221.328,A 0.000,B 0.000,C 90.000,E1 94.992} C_DIS
LIN {X 0.153,Y -571.237,Z 1221.326,A 0.000,B 0.000,C 90.000,E1 94.645} C_DIS
LIN {X -0.051,Y -567.372,Z 1221.325,A 0.000,B 0.000,C 90.000,E1 94.416} C_DIS
LIN {X -0.173,Y -564.449,Z 1221.322,A 0.000,B 0.000,C 90.000,E1 94.012} C_DIS
LIN {X 0.048,Y -564.342,Z 1221.321,A 0.000,B 0.000,C 90.000,E1 93.784} C_DIS
LIN {X -0.066,Y -564.543,Z 1221.315,A 0.000,B 0.000,C 90.000,E1 92.694} C_DIS
LIN {X 0.269,Y -565.993,Z 1221.303,A 0.000,B 0.000,C 90.000,E1 90.458} C_DIS
LIN {X -0.166,Y -567.166,Z 1221.294,A 0.000,B 0.000,C 90.000,E1 88.854} C_DIS
LIN {X 0.118,Y -568.570,Z 1221.283,A 0.000,B 0.000,C 90.000,E1 86.906} C_DIS
LIN {X -0.229,Y -569.878,Z 1221.274,A 0.000,B 0.000,C 90.000,E1 85.298} C_DIS
LIN {X 0.073,Y -571.310,Z 1221.265,A 0.000,B 0.000,C 90.000,E1 83.628} C_DIS
LIN {X -0.089,Y -572.774,Z 1221.256,A 0.000,B 0.000,C 90.000,E1 82.008} C_DIS
LIN {X -0.219,Y -574.140,Z 1221.247,A 0.000,B 0.000,C 90.000,E1 80.387} C_DIS
LIN {X -0.078,Y -574.863,Z 1221.240,A 0.000,B 0.000,C 90.000,E1 79.285} C_DIS
LIN {X -0.178,Y -575.717,Z 1221.233,A 0.000,B 0.000,C 90.000,E1 77.937} C_DIS
LIN {X 0.092,Y -576.385,Z 1221.227,A 0.000,B 0.000,C 90.000,E1 76.825} C_DIS
LIN {X 0.155,Y -577.125,Z 1221.219,A 0.000,B 0.000,C 90.000,E1 75.463} C_DIS
LIN {X 0.231,Y -577.858,Z 1221.212,A 0.000,B 0.000,C 90.000,E1 74.102} C_DIS
LIN {X -0.047,Y -578.894,Z 1221.201,A 0.000,B 0.000,C 90.000,E1 72.236} C_DIS
LIN {X 0.185,Y -579.373,Z 1221.197,A 0.000,B 0.000,C 90.000,E1 71.402} C_DIS
LIN {X 0.092,Y -580.182,Z 1221.189,A 0.000,B 0.000,C 90.000,E1 70.061} C_DIS
LIN {X -0.096,Y -581.656,Z 1221.177,A 0.000,B 0.000,C 90.000,E1 67.922} C_DIS
LIN {X -0.077,Y -583.020,Z 1221.168,A 0.000,B 0.000,C 90.000,E1 66.305} C_DIS
LIN {X -0.068,Y -584.083,Z 1221.162,A 0.000,B 0.000,C 90.000,E1 65.229} C_DIS
LIN {X 0.117,Y -585.745,Z 1221.152,A 0.000,B 0.000,C 90.000,E1 63.332} C_DIS
LIN {X 0.238,Y -587.920,Z 1221.140,A 0.000,B 0.000,C 90.000,E1 61.179} C_DIS
LIN {X -0.046,Y -589.311,Z 1221.133,A 0.000,B 0.000,C 90.000,E1 59.871} C_DIS
LIN {X 0.101,Y -590.389,Z 1221.127,A 0.000,B 0.000,C 90.000,E1 58.791} C_DIS
LIN {X 0.153,Y -591.624,Z 1221.119,A 0.000,B 0.000,C 90.000,E1 57.454} C_DIS
LIN {X 0.047,Y -592.724,Z 1221.112,A 0.000,B 0.000,C 90.000,E1 56.135} C_DIS
LIN {X -0.034,Y -593.830,Z 1221.105,A 0.000,B 0.000,C 90.000,E1 54.815} C_DIS
LIN {X -0.136,Y -595.249,Z 1221.094,A 0.000,B 0.000,C 90.000,E1 52.970} C_DIS
LIN {X 0.154,Y -596.607,Z 1221.084,A 0.000,B 0.000,C 90.000,E1 51.090} C_DIS
LIN {X -0.002,Y -597.075,Z 1221.080,A 0.000,B 0.000,C 90.000,E1 50.312} C_DIS
LIN {X 0.390,Y -597.998,Z 1221.068,A 0.000,B 0.000,C 90.000,E1 48.162} C_DIS
LIN {X 0.175,Y -598.276,Z 1221.063,A 0.000,B 0.000,C 90.000,E1 47.391} C_DIS
LIN {X 0.374,Y -598.658,Z 1221.056,A 0.000,B 0.000,C 90.000,E1 46.053} C_DIS
LIN {X -0.059,Y -598.693,Z 1221.050,A 0.000,B 0.000,C 90.000,E1 45.040} C_DIS
LIN {X 0.354,Y -598.543,Z 1221.044,A 0.000,B 0.000,C 90.000,E1 43.947} C_DIS
LIN {X 0.142,Y -598.300,Z 1221.040,A 0.000,B 0.000,C 90.000,E1 43.176} C_DIS
LIN {X 0.118,Y -597.469,Z 1221.031,A 0.000,B 0.000,C 90.000,E1 41.595} C_DIS
LIN {X 0.120,Y -597.236,Z 1221.028,A 0.000,B 0.000,C 90.000,E1 41.067} C_DIS
LIN {X -0.111,Y -596.403,Z 1221.021,A 0.000,B 0.000,C 90.000,E1 39.769} C_DIS
LIN {X -0.279,Y -595.383,Z 1221.014,A 0.000,B 0.000,C 90.000,E1 38.463} C_DIS
LIN {X -0.071,Y -594.626,Z 1221.009,A 0.000,B 0.000,C 90.000,E1 37.649} C_DIS
LIN {X -0.014,Y -593.297,Z 1221.003,A 0.000,B 0.000,C 90.000,E1 36.583} C_DIS
LIN {X -0.187,Y -592.187,Z 1220.999,A 0.000,B 0.000,C 90.000,E1 35.804} C_DIS
LIN {X -0.165,Y -590.462,Z 1220.993,A 0.000,B 0.000,C 90.000,E1 34.739} C_DIS
LIN {X -0.013,Y -588.265,Z 1220.987,A 0.000,B 0.000,C 90.000,E1 33.658} C_DIS
LIN {X 0.185,Y -587.686,Z 1220.986,A 0.000,B 0.000,C 90.000,E1 33.372} C_DIS
LIN {X -0.192,Y -584.722,Z 1220.980,A 0.000,B 0.000,C 90.000,E1 32.339} C_DIS
LIN {X -0.284,Y -582.354,Z 1220.975,A 0.000,B 0.000,C 90.000,E1 31.544} C_DIS
LIN {X -0.098,Y -579.374,Z 1220.971,A 0.000,B 0.000,C 90.000,E1 30.718} C_DIS
LIN {X 0.255,Y -576.081,Z 1220.966,A 0.000,B 0.000,C 90.000,E1 29.873} C_DIS
LIN {X 0.074,Y -572.320,Z 1220.962,A 0.000,B 0.000,C 90.000,E1 29.077} C_DIS
LIN {X -0.068,Y -568.798,Z 1220.958,A 0.000,B 0.000,C 90.000,E1 28.409} C_DIS
LIN {X 0.082,Y -565.764,Z 1220.955,A 0.000,B 0.000,C 90.000,E1 27.847} C_DIS
LIN {X -0.027,Y -562.542,Z 1220.952,A 0.000,B 0.000,C 90.000,E1 27.308} C_DIS
LIN {X 0.084,Y -559.126,Z 1220.949,A 0.000,B 0.000,C 90.000,E1 26.744} C_DIS
LIN {X 0.174,Y -555.494,Z 1220.946,A 0.000,B 0.000,C 90.000,E1 26.181} C_DIS
LIN {X -0.017,Y -551.600,Z 1220.943,A 0.000,B 0.000,C 90.000,E1 25.643} C_DIS
LIN {X 0.019,Y -547.391,Z 1220.939,A 0.000,B 0.000,C 90.000,E1 25.079} C_DIS
LIN {X -0.098,Y -541.777,Z 1220.935,A 0.000,B 0.000,C 90.000,E1 24.387} C_DIS
LIN {X 0.227,Y -535.768,Z 1220.932,A 0.000,B 0.000,C 90.000,E1 23.643} C_DIS
LIN {X -0.009,Y -527.000,Z 1220.926,A 0.000,B 0.000,C 90.000,E1 22.695} C_DIS
LIN {X 0.184,Y -520.436,Z 1220.922,A 0.000,B 0.000,C 90.000,E1 21.972} C_DIS
LIN {X -0.196,Y -511.034,Z 1220.917,A 0.000,B 0.000,C 90.000,E1 21.046} C_DIS
LIN {X -0.021,Y -499.944,Z 1220.911,A 0.000,B 0.000,C 90.000,E1 19.939} C_DIS
LIN {X -0.233,Y -489.939,Z 1220.906,A 0.000,B 0.000,C 90.000,E1 19.033} C_DIS
LIN {X -0.154,Y -482.675,Z 1220.902,A 0.000,B 0.000,C 90.000,E1 18.362} C_DIS
LIN {X 0.039,Y -474.092,Z 1220.898,A 0.000,B 0.000,C 90.000,E1 17.583} C_DIS
LIN {X -0.224,Y -458.289,Z 1220.890,A 0.000,B 0.000,C 90.000,E1 16.205} C_DIS
LIN {X -0.024,Y -440.599,Z 1220.881,A 0.000,B 0.000,C 90.000,E1 14.537} C_DIS
LIN {X 0.100,Y -420.582,Z 1220.870,A 0.000,B 0.000,C 90.000,E1 12.479} C_DIS
LIN {X 0.076,Y -402.713,Z 1220.858,A 0.000,B 0.000,C 90.000,E1 10.433} C_DIS
LIN {X 0.066,Y -397.834,Z 1220.854,A 0.000,B 0.000,C 90.000,E1 9.792} C_DIS
LIN {X 0.166,Y -394.614,Z 1220.852,A 0.000,B 0.000,C 90.000,E1 9.265} C_DIS
LIN {X 0.135,Y -393.654,Z 1220.850,A 0.000,B 0.000,C 90.000,E1 8.973} C_DIS
LIN {X 0.097,Y -393.647,Z 1220.850,A 0.000,B 0.000,C 90.000,E1 8.973} C_DIS
LIN {X 0.020,Y -393.848,Z 1220.849,A 0.000,B 0.000,C 90.000,E1 8.746} C_DIS
LIN {X -0.018,Y -393.870,Z 1220.849,A 0.000,B 0.000,C 90.000,E1 8.746} C_DIS
LIN {X -0.188,Y -396.547,Z 1220.845,A 0.000,B 0.000,C 90.000,E1 8.163} C_DIS
LIN {X -0.014,Y -397.064,Z 1220.845,A 0.000,B 0.000,C 90.000,E1 8.049} C_DIS
LIN {X -0.176,Y -400.641,Z 1220.842,A 0.000,B 0.000,C 90.000,E1 7.644} C_DIS
LIN {X 0.173,Y -405.888,Z 1220.840,A 0.000,B 0.000,C 90.000,E1 7.125} C_DIS
LIN {X -0.134,Y -420.076,Z 1220.834,A 0.000,B 0.000,C 90.000,E1 6.087} C_DIS
LIN {X -0.008,Y -431.257,Z 1220.829,A 0.000,B 0.000,C 90.000,E1 5.220} C_DIS
LIN {X 0.019,Y -443.944,Z 1220.824,A 0.000,B 0.000,C 90.000,E1 4.245} C_DIS
LIN {X 0.122,Y -456.605,Z 1220.818,A 0.000,B 0.000,C 90.000,E1 3.269} C_DIS
LIN {X -0.179,Y -465.957,Z 1220.814,A 0.000,B 0.000,C 90.000,E1 2.579} C_DIS
LIN {X 0.025,Y -472.084,Z 1220.812,A 0.000,B 0.000,C 90.000,E1 2.064} C_DIS
LIN {X -0.061,Y -479.405,Z 1220.808,A 0.000,B 0.000,C 90.000,E1 1.432} C_DIS
LIN {X -0.214,Y -485.199,Z 1220.805,A 0.000,B 0.000,C 90.000,E1 0.917} C_DIS
LIN {X -0.195,Y -492.045,Z 1220.801,A 0.000,B 0.000,C 90.000,E1 0.229} C_DIS
LIN {X 0.170,Y -498.487,Z 1220.797,A 0.000,B 0.000,C 90.000,E1 359.484} C_DIS
LIN {X 0.232,Y -504.769,Z 1220.793,A 0.000,B 0.000,C 90.000,E1 358.740} C_DIS
LIN {X -0.198,Y -510.535,Z 1220.789,A 0.000,B 0.000,C 90.000,E1 358.051} C_DIS
LIN {X -0.158,Y -515.859,Z 1220.785,A 0.000,B 0.000,C 90.000,E1 357.306} C_DIS
LIN {X -0.047,Y -520.828,Z 1220.781,A 0.000,B 0.000,C 90.000,E1 356.560} C_DIS
LIN {X -0.159,Y -524.542,Z 1220.778,A 0.000,B 0.000,C 90.000,E1 355.988} C_DIS
LIN {X 0.034,Y -528.755,Z 1220.774,A 0.000,B 0.000,C 90.000,E1 355.241} C_DIS
LIN {X 0.016,Y -531.854,Z 1220.770,A 0.000,B 0.000,C 90.000,E1 354.666} C_DIS
LIN {X 0.059,Y -535.970,Z 1220.766,A 0.000,B 0.000,C 90.000,E1 353.799} C_DIS
LIN {X -0.168,Y -537.940,Z 1220.763,A 0.000,B 0.000,C 90.000,E1 353.394} C_DIS
LIN {X -0.053,Y -541.431,Z 1220.759,A 0.000,B 0.000,C 90.000,E1 352.527} C_DIS
LIN {X 0.018,Y -543.649,Z 1220.755,A 0.000,B 0.000,C 90.000,E1 351.951} C_DIS
LIN {X 0.189,Y -546.608,Z 1220.751,A 0.000,B 0.000,C 90.000,E1 351.084} C_DIS
LIN {X -0.153,Y -549.322,Z 1220.746,A 0.000,B 0.000,C 90.000,E1 350.274} C_DIS
LIN {X -0.142,Y -553.282,Z 1220.738,A 0.000,B 0.000,C 90.000,E1 348.870} C_DIS
LIN {X -0.186,Y -556.185,Z 1220.732,A 0.000,B 0.000,C 90.000,E1 347.757} C_DIS
LIN {X -0.191,Y -558.753,Z 1220.726,A 0.000,B 0.000,C 90.000,E1 346.645} C_DIS
LIN {X 0.115,Y -561.674,Z 1220.718,A 0.000,B 0.000,C 90.000,E1 345.227} C_DIS
LIN {X 0.166,Y -563.302,Z 1220.713,A 0.000,B 0.000,C 90.000,E1 344.393} C_DIS
LIN {X -0.152,Y -565.320,Z 1220.707,A 0.000,B 0.000,C 90.000,E1 343.323} C_DIS
LIN {X 0.261,Y -567.062,Z 1220.701,A 0.000,B 0.000,C 90.000,E1 342.181} C_DIS
LIN {X -0.224,Y -568.975,Z 1220.694,A 0.000,B 0.000,C 90.000,E1 340.859} C_DIS
LIN {X 0.077,Y -569.962,Z 1220.689,A 0.000,B 0.000,C 90.000,E1 340.007} C_DIS
LIN {X -0.146,Y -570.702,Z 1220.684,A 0.000,B 0.000,C 90.000,E1 339.209} C_DIS
LIN {X 0.171,Y -571.203,Z 1220.680,A 0.000,B 0.000,C 90.000,E1 338.358} C_DIS
LIN {X 0.004,Y -571.446,Z 1220.674,A 0.000,B 0.000,C 90.000,E1 337.283} C_DIS
LIN {X 0.148,Y -571.130,Z 1220.668,A 0.000,B 0.000,C 90.000,E1 336.177} C_DIS
LIN {X 0.161,Y -570.459,Z 1220.663,A 0.000,B 0.000,C 90.000,E1 335.357} C_DIS
LIN {X -0.005,Y -569.113,Z 1220.657,A 0.000,B 0.000,C 90.000,E1 334.280} C_DIS
LIN {X 0.159,Y -568.153,Z 1220.654,A 0.000,B 0.000,C 90.000,E1 333.717} C_DIS
LIN {X -0.115,Y -566.424,Z 1220.650,A 0.000,B 0.000,C 90.000,E1 332.922} C_DIS
LIN {X -0.158,Y -564.380,Z 1220.645,A 0.000,B 0.000,C 90.000,E1 332.103} C_DIS
LIN {X 0.227,Y -562.850,Z 1220.642,A 0.000,B 0.000,C 90.000,E1 331.513} C_DIS
LIN {X 0.112,Y -560.912,Z 1220.639,A 0.000,B 0.000,C 90.000,E1 330.973} C_DIS
LIN {X -0.287,Y -558.666,Z 1220.636,A 0.000,B 0.000,C 90.000,E1 330.461} C_DIS
LIN {X 0.162,Y -556.759,Z 1220.633,A 0.000,B 0.000,C 90.000,E1 329.999} C_DIS
LIN {X 0.009,Y -553.929,Z 1220.630,A 0.000,B 0.000,C 90.000,E1 329.459} C_DIS
LIN {X 0.193,Y -550.022,Z 1220.626,A 0.000,B 0.000,C 90.000,E1 328.742} C_DIS
LIN {X 0.029,Y -544.569,Z 1220.622,A 0.000,B 0.000,C 90.000,E1 327.916} C_DIS
LIN {X -0.072,Y -541.677,Z 1220.620,A 0.000,B 0.000,C 90.000,E1 327.502} C_DIS
LIN {X -0.013,Y -536.208,Z 1220.615,A 0.000,B 0.000,C 90.000,E1 326.786} C_DIS
LIN {X -0.178,Y -528.327,Z 1220.610,A 0.000,B 0.000,C 90.000,E1 325.801} C_DIS
LIN {X -0.050,Y -518.006,Z 1220.603,A 0.000,B 0.000,C 90.000,E1 324.482} C_DIS
LIN {X -0.301,Y -514.534,Z 1220.600,A 0.000,B 0.000,C 90.000,E1 323.989} C_DIS
LIN {X 0.269,Y -511.680,Z 1220.597,A 0.000,B 0.000,C 90.000,E1 323.417} C_DIS
LIN {X -0.056,Y -509.598,Z 1220.594,A 0.000,B 0.000,C 90.000,E1 322.844} C_DIS
LIN {X -0.032,Y -508.733,Z 1220.591,A 0.000,B 0.000,C 90.000,E1 322.396} C_DIS
LIN {X -0.122,Y -508.341,Z 1220.589,A 0.000,B 0.000,C 90.000,E1 322.110} C_DIS
LIN {X -0.308,Y -507.952,Z 1220.586,A 0.000,B 0.000,C 90.000,E1 321.537} C_DIS
LIN {X 0.114,Y -507.827,Z 1220.581,A 0.000,B 0.000,C 90.000,E1 320.598} C_DIS
LIN {X 0.157,Y -509.339,Z 1220.566,A 0.000,B 0.000,C 90.000,E1 317.919} C_DIS
LIN {X -0.041,Y -510.171,Z 1220.558,A 0.000,B 0.000,C 90.000,E1 316.458} C_DIS
LIN {X -0.244,Y -510.926,Z 1220.550,A 0.000,B 0.000,C 90.000,E1 315.000} C_DIS
LIN {X -0.183,Y -511.713,Z 1220.540,A 0.000,B 0.000,C 90.000,E1 313.218} C_DIS
LIN {X -0.089,Y -512.564,Z 1220.530,A 0.000,B 0.000,C 90.000,E1 311.434} C_DIS
LIN {X 0.155,Y -513.259,Z 1220.522,A 0.000,B 0.000,C 90.000,E1 309.930} C_DIS
LIN {X 0.164,Y -513.728,Z 1220.515,A 0.000,B 0.000,C 90.000,E1 308.749} C_DIS
LIN {X -0.123,Y -514.514,Z 1220.502,A 0.000,B 0.000,C 90.000,E1 306.423} C_DIS
LIN {X 0.206,Y -515.280,Z 1220.491,A 0.000,B 0.000,C 90.000,E1 304.326} C_DIS
LIN {X -0.018,Y -515.801,Z 1220.483,A 0.000,B 0.000,C 90.000,E1 302.880} C_DIS
LIN {X -0.072,Y -516.150,Z 1220.474,A 0.000,B 0.000,C 90.000,E1 301.416} C_DIS
LIN {X 0.148,Y -516.392,Z 1220.466,A 0.000,B 0.000,C 90.000,E1 299.922} C_DIS
LIN {X -0.150,Y -516.541,Z 1220.458,A 0.000,B 0.000,C 90.000,E1 298.487} C_DIS
LIN {X 0.013,Y -516.693,Z 1220.450,A 0.000,B 0.000,C 90.000,E1 297.001} C_DIS
LIN {X -0.052,Y -516.738,Z 1220.442,A 0.000,B 0.000,C 90.000,E1 295.540} C_DIS
LIN {X -0.116,Y -516.851,Z 1220.434,A 0.000,B 0.000,C 90.000,E1 294.079} C_DIS
LIN {X -0.259,Y -516.884,Z 1220.424,A 0.000,B 0.000,C 90.000,E1 292.333} C_DIS
LIN {X 0.282,Y -516.706,Z 1220.417,A 0.000,B 0.000,C 90.000,E1 291.099} C_DIS
LIN {X 0.019,Y -516.372,Z 1220.413,A 0.000,B 0.000,C 90.000,E1 290.248} C_DIS
LIN {X 0.101,Y -515.414,Z 1220.401,A 0.000,B 0.000,C 90.000,E1 288.181} C_DIS
LIN {X -0.127,Y -514.582,Z 1220.391,A 0.000,B 0.000,C 90.000,E1 286.441} C_DIS
LIN {X 0.007,Y -513.721,Z 1220.383,A 0.000,B 0.000,C 90.000,E1 284.954} C_DIS
LIN {X 0.088,Y -512.666,Z 1220.373,A 0.000,B 0.000,C 90.000,E1 283.175} C_DIS
LIN {X -0.028,Y -511.901,Z 1220.367,A 0.000,B 0.000,C 90.000,E1 282.007} C_DIS
LIN {X -0.184,Y -510.848,Z 1220.359,A 0.000,B 0.000,C 90.000,E1 280.546} C_DIS
LIN {X 0.019,Y -509.700,Z 1220.349,A 0.000,B 0.000,C 90.000,E1 278.746} C_DIS
LIN {X -0.085,Y -508.010,Z 1220.334,A 0.000,B 0.000,C 90.000,E1 276.087} C_DIS
LIN {X -0.144,Y -506.817,Z 1220.322,A 0.000,B 0.000,C 90.000,E1 274.012} C_DIS
LIN {X 0.078,Y -506.341,Z 1220.317,A 0.000,B 0.000,C 90.000,E1 273.094} C_DIS
LIN {X -0.131,Y -505.024,Z 1220.306,A 0.000,B 0.000,C 90.000,E1 271.031} C_DIS
LIN {X 0.017,Y -503.603,Z 1220.292,A 0.000,B 0.000,C 90.000,E1 268.625} C_DIS
LIN {X -0.235,Y -502.392,Z 1220.281,A 0.000,B 0.000,C 90.000,E1 266.560} C_DIS
LIN {X -0.184,Y -501.617,Z 1220.274,A 0.000,B 0.000,C 90.000,E1 265.355} C_DIS
LIN {X 0.171,Y -500.270,Z 1220.264,A 0.000,B 0.000,C 90.000,E1 263.514} C_DIS
LIN {X 0.204,Y -498.932,Z 1220.256,A 0.000,B 0.000,C 90.000,E1 262.008} C_DIS
LIN {X -0.033,Y -497.038,Z 1220.244,A 0.000,B 0.000,C 90.000,E1 259.926} C_DIS
LIN {X -0.052,Y -495.218,Z 1220.232,A 0.000,B 0.000,C 90.000,E1 257.813} C_DIS
LIN {X -0.107,Y -493.667,Z 1220.221,A 0.000,B 0.000,C 90.000,E1 255.700} C_DIS
LIN {X 0.088,Y -492.808,Z 1220.214,A 0.000,B 0.000,C 90.000,E1 254.464} C_DIS
LIN {X -0.221,Y -491.348,Z 1220.199,A 0.000,B 0.000,C 90.000,E1 251.764} C_DIS
LIN {X -0.219,Y -490.627,Z 1220.190,A 0.000,B 0.000,C 90.000,E1 250.242} C_DIS
LIN {X -0.119,Y -490.198,Z 1220.185,A 0.000,B 0.000,C 90.000,E1 249.316} C_DIS
LIN {X -0.140,Y -489.280,Z 1220.177,A 0.000,B 0.000,C 90.000,E1 247.794} C_DIS
LIN {X 0.185,Y -488.127,Z 1220.168,A 0.000,B 0.000,C 90.000,E1 246.230} C_DIS
LIN {X 0.060,Y -486.458,Z 1220.158,A 0.000,B 0.000,C 90.000,E1 244.409} C_DIS
LIN {X 0.094,Y -484.914,Z 1220.149,A 0.000,B 0.000,C 90.000,E1 242.871} C_DIS
LIN {X -0.117,Y -483.966,Z 1220.144,A 0.000,B 0.000,C 90.000,E1 241.975} C_DIS
LIN {X 0.109,Y -482.551,Z 1220.137,A 0.000,B 0.000,C 90.000,E1 240.717} C_DIS
LIN {X 0.074,Y -481.099,Z 1220.131,A 0.000,B 0.000,C 90.000,E1 239.488} C_DIS
LIN {X 0.094,Y -479.717,Z 1220.124,A 0.000,B 0.000,C 90.000,E1 238.250} C_DIS
LIN {X -0.158,Y -477.486,Z 1220.113,A 0.000,B 0.000,C 90.000,E1 236.421} C_DIS
LIN {X 0.072,Y -475.364,Z 1220.103,A 0.000,B 0.000,C 90.000,E1 234.529} C_DIS
LIN {X -0.130,Y -473.383,Z 1220.093,A 0.000,B 0.000,C 90.000,E1 232.683} C_DIS
LIN {X -0.032,Y -470.291,Z 1220.075,A 0.000,B 0.000,C 90.000,E1 229.542} C_DIS
LIN {X 0.085,Y -468.881,Z 1220.067,A 0.000,B 0.000,C 90.000,E1 227.957} C_DIS
LIN {X 0.213,Y -467.133,Z 1220.056,A 0.000,B 0.000,C 90.000,E1 226.053} C_DIS
LIN {X 0.057,Y -464.124,Z 1220.017,A 0.000,B 0.000,C 90.000,E1 219.116} C_DIS
LIN {X -0.061,Y -464.988,Z 1220.000,A 0.000,B 0.000,C 90.000,E1 215.964} C_DIS
LIN {X 0.105,Y -466.895,Z 1219.980,A 0.000,B 0.000,C 90.000,E1 212.467} C_DIS
LIN {X -0.017,Y -468.621,Z 1219.970,A 0.000,B 0.000,C 90.000,E1 210.590} C_DIS
LIN {X -0.124,Y -472.044,Z 1219.953,A 0.000,B 0.000,C 90.000,E1 207.462} C_DIS
LIN {X -0.208,Y -474.705,Z 1219.940,A 0.000,B 0.000,C 90.000,E1 205.283} C_DIS
LIN {X -0.073,Y -480.896,Z 1219.918,A 0.000,B 0.000,C 90.000,E1 201.227} C_DIS
LIN {X 0.115,Y -488.380,Z 1219.897,A 0.000,B 0.000,C 90.000,E1 197.511} C_DIS
LIN {X 0.012,Y -496.601,Z 1219.879,A 0.000,B 0.000,C 90.000,E1 194.175} C_DIS
LIN {X -0.030,Y -503.244,Z 1219.865,A 0.000,B 0.000,C 90.000,E1 191.771} C_DIS
LIN {X 0.121,Y -508.240,Z 1219.855,A 0.000,B 0.000,C 90.000,E1 189.962} C_DIS
LIN {X -0.210,Y -513.565,Z 1219.846,A 0.000,B 0.000,C 90.000,E1 188.219} C_DIS
LIN {X 0.115,Y -517.142,Z 1219.839,A 0.000,B 0.000,C 90.000,E1 187.004} C_DIS
LIN {X -0.082,Y -520.612,Z 1219.833,A 0.000,B 0.000,C 90.000,E1 185.853} C_DIS
LIN {X 0.193,Y -526.612,Z 1219.821,A 0.000,B 0.000,C 90.000,E1 183.784} C_DIS
LIN {X 0.056,Y -531.814,Z 1219.812,A 0.000,B 0.000,C 90.000,E1 182.064} C_DIS
LIN {X 0.039,Y -537.766,Z 1219.800,A 0.000,B 0.000,C 90.000,E1 180.057} C_DIS
LIN {X 0.090,Y -541.089,Z 1219.794,A 0.000,B 0.000,C 90.000,E1 178.912} C_DIS
LIN {X 0.233,Y -545.211,Z 1219.786,A 0.000,B 0.000,C 90.000,E1 177.478} C_DIS
LIN {X -0.098,Y -549.098,Z 1219.778,A 0.000,B 0.000,C 90.000,E1 176.102} C_DIS
LIN {X -0.226,Y -553.631,Z 1219.769,A 0.000,B 0.000,C 90.000,E1 174.432} C_DIS
LIN {X -0.254,Y -557.984,Z 1219.760,A 0.000,B 0.000,C 90.000,E1 172.761} C_DIS
LIN {X -0.272,Y -561.564,Z 1219.752,A 0.000,B 0.000,C 90.000,E1 171.376} C_DIS
LIN {X -0.145,Y -565.119,Z 1219.744,A 0.000,B 0.000,C 90.000,E1 169.982} C_DIS
LIN {X -0.043,Y -569.977,Z 1219.734,A 0.000,B 0.000,C 90.000,E1 168.049} C_DIS
LIN {X -0.210,Y -573.510,Z 1219.726,A 0.000,B 0.000,C 90.000,E1 166.700} C_DIS
LIN {X 0.233,Y -578.679,Z 1219.715,A 0.000,B 0.000,C 90.000,E1 164.755} C_DIS
LIN {X 0.118,Y -586.438,Z 1219.701,A 0.000,B 0.000,C 90.000,E1 162.072} C_DIS
LIN {X 0.148,Y -593.369,Z 1219.689,A 0.000,B 0.000,C 90.000,E1 159.934} C_DIS
LIN {X 0.309,Y -602.091,Z 1219.675,A 0.000,B 0.000,C 90.000,E1 157.539} C_DIS
LIN {X 0.295,Y -606.994,Z 1219.668,A 0.000,B 0.000,C 90.000,E1 156.230} C_DIS
LIN {X -0.232,Y -612.744,Z 1219.659,A 0.000,B 0.000,C 90.000,E1 154.717} C_DIS
LIN {X 0.231,Y -615.541,Z 1219.655,A 0.000,B 0.000,C 90.000,E1 153.896} C_DIS
LIN {X 0.154,Y -619.120,Z 1219.649,A 0.000,B 0.000,C 90.000,E1 152.871} C_DIS
LIN {X 0.120,Y -623.428,Z 1219.642,A 0.000,B 0.000,C 90.000,E1 151.591} C_DIS
LIN {X -0.097,Y -627.657,Z 1219.635,A 0.000,B 0.000,C 90.000,E1 150.333} C_DIS
LIN {X 0.108,Y -632.590,Z 1219.627,A 0.000,B 0.000,C 90.000,E1 148.791} C_DIS
LIN {X -0.120,Y -637.340,Z 1219.618,A 0.000,B 0.000,C 90.000,E1 147.296} C_DIS
LIN {X -0.260,Y -641.710,Z 1219.610,A 0.000,B 0.000,C 90.000,E1 145.801} C_DIS
LIN {X 0.062,Y -643.711,Z 1219.606,A 0.000,B 0.000,C 90.000,E1 145.022} C_DIS
LIN {X -0.070,Y -646.263,Z 1219.600,A 0.000,B 0.000,C 90.000,E1 144.036} C_DIS
LIN {X -0.173,Y -648.566,Z 1219.595,A 0.000,B 0.000,C 90.000,E1 143.050} C_DIS
LIN {X 0.115,Y -651.987,Z 1219.586,A 0.000,B 0.000,C 90.000,E1 141.537} C_DIS
LIN {X 0.005,Y -654.698,Z 1219.580,A 0.000,B 0.000,C 90.000,E1 140.312} C_DIS
LIN {X -0.153,Y -657.367,Z 1219.573,A 0.000,B 0.000,C 90.000,E1 139.094} C_DIS
LIN {X -0.290,Y -660.638,Z 1219.565,A 0.000,B 0.000,C 90.000,E1 137.634} C_DIS
LIN {X 0.067,Y -664.857,Z 1219.554,A 0.000,B 0.000,C 90.000,E1 135.648} C_DIS
LIN {X 0.061,Y -668.923,Z 1219.544,A 0.000,B 0.000,C 90.000,E1 133.947} C_DIS
LIN {X 0.173,Y -673.203,Z 1219.535,A 0.000,B 0.000,C 90.000,E1 132.243} C_DIS
LIN {X -0.175,Y -676.219,Z 1219.528,A 0.000,B 0.000,C 90.000,E1 131.067} C_DIS
LIN {X 0.171,Y -680.415,Z 1219.519,A 0.000,B 0.000,C 90.000,E1 129.358} C_DIS
LIN {X 0.006,Y -683.385,Z 1219.512,A 0.000,B 0.000,C 90.000,E1 128.177} C_DIS
LIN {X 0.051,Y -687.018,Z 1219.504,A 0.000,B 0.000,C 90.000,E1 126.744} C_DIS
LIN {X -0.066,Y -689.317,Z 1219.499,A 0.000,B 0.000,C 90.000,E1 125.804} C_DIS
LIN {X -0.318,Y -692.600,Z 1219.491,A 0.000,B 0.000,C 90.000,E1 124.405} C_DIS
LIN {X -0.166,Y -695.194,Z 1219.484,A 0.000,B 0.000,C 90.000,E1 123.214} C_DIS
LIN {X -0.017,Y -697.250,Z 1219.479,A 0.000,B 0.000,C 90.000,E1 122.260} C_DIS
LIN {X 0.051,Y -699.605,Z 1219.473,A 0.000,B 0.000,C 90.000,E1 121.082} C_DIS
LIN {X 0.258,Y -701.399,Z 1219.468,A 0.000,B 0.000,C 90.000,E1 120.129} C_DIS
LIN {X -0.210,Y -703.502,Z 1219.461,A 0.000,B 0.000,C 90.000,E1 118.999} C_DIS
LIN {X 0.299,Y -704.950,Z 1219.456,A 0.000,B 0.000,C 90.000,E1 118.025} C_DIS
LIN {X 0.213,Y -705.685,Z 1219.452,A 0.000,B 0.000,C 90.000,E1 117.334} C_DIS
LIN {X 0.120,Y -706.320,Z 1219.447,A 0.000,B 0.000,C 90.000,E1 116.411} C_DIS
LIN {X 0.055,Y -706.576,Z 1219.443,A 0.000,B 0.000,C 90.000,E1 115.720} C_DIS
LIN {X -0.004,Y -706.450,Z 1219.439,A 0.000,B 0.000,C 90.000,E1 115.027} C_DIS
LIN {X -0.062,Y -706.115,Z 1219.437,A 0.000,B 0.000,C 90.000,E1 114.567} C_DIS
LIN {X 0.227,Y -705.209,Z 1219.434,A 0.000,B 0.000,C 90.000,E1 114.079} C_DIS
LIN {X -0.129,Y -704.630,Z 1219.433,A 0.000,B 0.000,C 90.000,E1 113.875} C_DIS
LIN {X 0.155,Y -702.558,Z 1219.430,A 0.000,B 0.000,C 90.000,E1 113.387} C_DIS
LIN {X 0.293,Y -701.937,Z 1219.429,A 0.000,B 0.000,C 90.000,E1 113.259} C_DIS
LIN {X 0.156,Y -701.009,Z 1219.429,A 0.000,B 0.000,C 90.000,E1 113.153} C_DIS
LIN {X 0.067,Y -696.873,Z 1219.427,A 0.000,B 0.000,C 90.000,E1 112.823} C_DIS
LIN {X 0.078,Y -695.575,Z 1219.426,A 0.000,B 0.000,C 90.000,E1 112.717} C_DIS
LIN {X -0.292,Y -694.026,Z 1219.426,A 0.000,B 0.000,C 90.000,E1 112.642} C_DIS
LIN {X -0.022,Y -691.381,Z 1219.425,A 0.000,B 0.000,C 90.000,E1 112.514} C_DIS
LIN {X 0.072,Y -685.947,Z 1219.424,A 0.000,B 0.000,C 90.000,E1 112.333} C_DIS
LIN {X -0.256,Y -683.798,Z 1219.424,A 0.000,B 0.000,C 90.000,E1 112.333} C_DIS
LIN {X 0.048,Y -677.077,Z 1219.424,A 0.000,B 0.000,C 90.000,E1 112.280} C_DIS
LIN {X -0.001,Y -613.024,Z 1219.424,A 0.000,B 0.000,C 90.000,E1 112.280} C_DIS
LIN {X -0.207,Y -611.157,Z 1219.423,A 0.000,B 0.000,C 90.000,E1 112.206} C_DIS
LIN {X 0.038,Y -607.047,Z 1219.422,A 0.000,B 0.000,C 90.000,E1 111.897} C_DIS
LIN {X 0.129,Y -603.364,Z 1219.420,A 0.000,B 0.000,C 90.000,E1 111.535} C_DIS
LIN {X 0.152,Y -602.318,Z 1219.419,A 0.000,B 0.000,C 90.000,E1 111.408} C_DIS
LIN {X 0.035,Y -601.703,Z 1219.418,A 0.000,B 0.000,C 90.000,E1 111.280} C_DIS
LIN {X -0.094,Y -601.531,Z 1219.418,A 0.000,B 0.000,C 90.000,E1 111.227} C_DIS
LIN {X -0.260,Y -601.808,Z 1219.417,A 0.000,B 0.000,C 90.000,E1 111.046} C_DIS
LIN {X 0.246,Y -603.339,Z 1219.414,A 0.000,B 0.000,C 90.000,E1 110.482} C_DIS
LIN {X 0.090,Y -607.160,Z 1219.408,A 0.000,B 0.000,C 90.000,E1 109.450} C_DIS
LIN {X -0.018,Y -610.556,Z 1219.402,A 0.000,B 0.000,C 90.000,E1 108.417} C_DIS
LIN {X -0.232,Y -616.788,Z 1219.392,A 0.000,B 0.000,C 90.000,E1 106.622} C_DIS
LIN {X -0.168,Y -619.403,Z 1219.388,A 0.000,B 0.000,C 90.000,E1 105.843} C_DIS
LIN {X 0.202,Y -620.247,Z 1219.387,A 0.000,B 0.000,C 90.000,E1 105.552} C_DIS
LIN {X 0.299,Y -622.279,Z 1219.382,A 0.000,B 0.000,C 90.000,E1 104.773} C_DIS
LIN {X -0.135,Y -623.418,Z 1219.379,A 0.000,B 0.000,C 90.000,E1 104.300} C_DIS
LIN {X -0.164,Y -624.719,Z 1219.375,A 0.000,B 0.000,C 90.000,E1 103.536} C_DIS
LIN {X 0.027,Y -625.280,Z 1219.372,A 0.000,B 0.000,C 90.000,E1 103.008} C_DIS
LIN {X 0.225,Y -625.283,Z 1219.370,A 0.000,B 0.000,C 90.000,E1 102.479} C_DIS
LIN {X -0.188,Y -625.004,Z 1219.367,A 0.000,B 0.000,C 90.000,E1 102.007} C_DIS
LIN {X 0.215,Y -624.775,Z 1219.365,A 0.000,B 0.000,C 90.000,E1 101.715} C_DIS
LIN {X -0.205,Y -623.946,Z 1219.362,A 0.000,B 0.000,C 90.000,E1 101.243} C_DIS
LIN {X -0.020,Y -622.796,Z 1219.360,A 0.000,B 0.000,C 90.000,E1 100.715} C_DIS
LIN {X 0.043,Y -621.306,Z 1219.357,A 0.000,B 0.000,C 90.000,E1 100.197} C_DIS
LIN {X -0.179,Y -620.417,Z 1219.355,A 0.000,B 0.000,C 90.000,E1 99.962} C_DIS
LIN {X 0.255,Y -617.082,Z 1219.351,A 0.000,B 0.000,C 90.000,E1 99.151} C_DIS
LIN {X 0.019,Y -615.888,Z 1219.350,A 0.000,B 0.000,C 90.000,E1 98.916} C_DIS
LIN {X 0.044,Y -612.670,Z 1219.347,A 0.000,B 0.000,C 90.000,E1 98.398} C_DIS
LIN {X -0.041,Y -607.695,Z 1219.343,A 0.000,B 0.000,C 90.000,E1 97.757} C_DIS
LIN {X -0.066,Y -602.880,Z 1219.340,A 0.000,B 0.000,C 90.000,E1 97.239} C_DIS
LIN {X 0.108,Y -597.622,Z 1219.337,A 0.000,B 0.000,C 90.000,E1 96.720} C_DIS
LIN {X -0.030,Y -591.992,Z 1219.335,A 0.000,B 0.000,C 90.000,E1 96.258} C_DIS
LIN {X 0.074,Y -587.263,Z 1219.333,A 0.000,B 0.000,C 90.000,E1 95.910} C_DIS
LIN {X -0.168,Y -582.638,Z 1219.331,A 0.000,B 0.000,C 90.000,E1 95.625} C_DIS
LIN {X 0.156,Y -575.937,Z 1219.329,A 0.000,B 0.000,C 90.000,E1 95.220} C_DIS
LIN {X -0.175,Y -571.070,Z 1219.328,A 0.000,B 0.000,C 90.000,E1 94.992} C_DIS
LIN {X -0.208,Y -567.356,Z 1219.326,A 0.000,B 0.000,C 90.000,E1 94.759} C_DIS
LIN {X -0.032,Y -566.674,Z 1219.326,A 0.000,B 0.000,C 90.000,E1 94.645} C_DIS
LIN {X -0.262,Y -564.169,Z 1219.323,A 0.000,B 0.000,C 90.000,E1 94.188} C_DIS
LIN {X 0.259,Y -564.147,Z 1219.323,A 0.000,B 0.000,C 90.000,E1 94.131} C_DIS
LIN {X -0.234,Y -564.016,Z 1219.321,A 0.000,B 0.000,C 90.000,E1 93.841} C_DIS
LIN {X 0.212,Y -564.413,Z 1219.315,A 0.000,B 0.000,C 90.000,E1 92.694} C_DIS
LIN {X -0.135,Y -565.725,Z 1219.304,A 0.000,B 0.000,C 90.000,E1 90.802} C_DIS
LIN {X -0.010,Y -566.885,Z 1219.295,A 0.000,B 0.000,C 90.000,E1 89.141} C_DIS
LIN {X 0.033,Y -567.885,Z 1219.288,A 0.000,B 0.000,C 90.000,E1 87.764} C_DIS
LIN {X -0.196,Y -569.364,Z 1219.277,A 0.000,B 0.000,C 90.000,E1 85.869} C_DIS
LIN {X -0.225,Y -571.209,Z 1219.265,A 0.000,B 0.000,C 90.000,E1 83.685} C_DIS
LIN {X 0.179,Y -572.650,Z 1219.256,A 0.000,B 0.000,C 90.000,E1 82.008} C_DIS
LIN {X 0.047,Y -573.979,Z 1219.247,A 0.000,B 0.000,C 90.000,E1 80.387} C_DIS
LIN {X -0.175,Y -574.885,Z 1219.239,A 0.000,B 0.000,C 90.000,E1 79.050} C_DIS
LIN {X 0.084,Y -575.565,Z 1219.233,A 0.000,B 0.000,C 90.000,E1 77.937} C_DIS
LIN {X -0.209,Y -576.228,Z 1219.227,A 0.000,B 0.000,C 90.000,E1 76.881} C_DIS
LIN {X -0.146,Y -576.959,Z 1219.219,A 0.000,B 0.000,C 90.000,E1 75.519} C_DIS
LIN {X -0.070,Y -577.687,Z 1219.212,A 0.000,B 0.000,C 90.000,E1 74.157} C_DIS
LIN {X 0.204,Y -578.705,Z 1219.201,A 0.000,B 0.000,C 90.000,E1 72.236} C_DIS
LIN {X -0.116,Y -579.197,Z 1219.197,A 0.000,B 0.000,C 90.000,E1 71.456} C_DIS
LIN {X -0.207,Y -579.993,Z 1219.189,A 0.000,B 0.000,C 90.000,E1 70.115} C_DIS
LIN {X 0.147,Y -581.486,Z 1219.177,A 0.000,B 0.000,C 90.000,E1 67.922} C_DIS
LIN {X 0.162,Y -582.855,Z 1219.168,A 0.000,B 0.000,C 90.000,E1 66.305} C_DIS
LIN {X 0.170,Y -583.924,Z 1219.162,A 0.000,B 0.000,C 90.000,E1 65.229} C_DIS
LIN {X -0.173,Y -585.593,Z 1219.152,A 0.000,B 0.000,C 90.000,E1 63.384} C_DIS
LIN {X -0.212,Y -587.500,Z 1219.142,A 0.000,B 0.000,C 90.000,E1 61.513} C_DIS
LIN {X 0.182,Y -589.160,Z 1219.133,A 0.000,B 0.000,C 90.000,E1 59.871} C_DIS
LIN {X 0.213,Y -590.442,Z 1219.125,A 0.000,B 0.000,C 90.000,E1 58.535} C_DIS
LIN {X -0.122,Y -591.449,Z 1219.119,A 0.000,B 0.000,C 90.000,E1 57.502} C_DIS
LIN {X -0.061,Y -592.546,Z 1219.112,A 0.000,B 0.000,C 90.000,E1 56.167} C_DIS
LIN {X 0.183,Y -593.643,Z 1219.105,A 0.000,B 0.000,C 90.000,E1 54.815} C_DIS
LIN {X 0.079,Y -595.053,Z 1219.094,A 0.000,B 0.000,C 90.000,E1 52.970} C_DIS
LIN {X 0.136,Y -596.210,Z 1219.086,A 0.000,B 0.000,C 90.000,E1 51.376} C_DIS
LIN {X -0.253,Y -596.893,Z 1219.080,A 0.000,B 0.000,C 90.000,E1 50.356} C_DIS
LIN {X -0.028,Y -597.706,Z 1219.069,A 0.000,B 0.000,C 90.000,E1 48.485} C_DIS
LIN {X 0.376,Y -598.068,Z 1219.063,A 0.000,B 0.000,C 90.000,E1 47.391} C_DIS
LIN {X 0.357,Y -598.518,Z 1219.055,A 0.000,B 0.000,C 90.000,E1 45.810} C_DIS
LIN {X 0.130,Y -598.455,Z 1219.047,A 0.000,B 0.000,C 90.000,E1 44.514} C_DIS
LIN {X 0.114,Y -598.236,Z 1219.042,A 0.000,B 0.000,C 90.000,E1 43.461} C_DIS
LIN {X -0.317,Y -597.414,Z 1219.033,A 0.000,B 0.000,C 90.000,E1 41.919} C_DIS
LIN {X 0.305,Y -597.038,Z 1219.028,A 0.000,B 0.000,C 90.000,E1 41.067} C_DIS
LIN {X 0.070,Y -596.173,Z 1219.021,A 0.000,B 0.000,C 90.000,E1 39.769} C_DIS
LIN {X -0.102,Y -595.133,Z 1219.014,A 0.000,B 0.000,C 90.000,E1 38.463} C_DIS
LIN {X 0.103,Y -594.386,Z 1219.009,A 0.000,B 0.000,C 90.000,E1 37.649} C_DIS
LIN {X 0.157,Y -593.057,Z 1219.003,A 0.000,B 0.000,C 90.000,E1 36.583} C_DIS
LIN {X -0.236,Y -592.373,Z 1219.000,A 0.000,B 0.000,C 90.000,E1 36.091} C_DIS
LIN {X 0.000,Y -590.220,Z 1218.993,A 0.000,B 0.000,C 90.000,E1 34.739} C_DIS
LIN {X 0.147,Y -588.003,Z 1218.987,A 0.000,B 0.000,C 90.000,E1 33.658} C_DIS
LIN {X -0.147,Y -587.429,Z 1218.986,A 0.000,B 0.000,C 90.000,E1 33.420} C_DIS
LIN {X -0.219,Y -585.210,Z 1218.981,A 0.000,B 0.000,C 90.000,E1 32.625} C_DIS
LIN {X -0.132,Y -582.062,Z 1218.975,A 0.000,B 0.000,C 90.000,E1 31.544} C_DIS
LIN {X 0.049,Y -579.065,Z 1218.971,A 0.000,B 0.000,C 90.000,E1 30.718} C_DIS
LIN {X -0.102,Y -575.756,Z 1218.966,A 0.000,B 0.000,C 90.000,E1 29.922} C_DIS
LIN {X 0.092,Y -573.267,Z 1218.963,A 0.000,B 0.000,C 90.000,E1 29.361} C_DIS
LIN {X -0.119,Y -569.202,Z 1218.959,A 0.000,B 0.000,C 90.000,E1 28.565} C_DIS
LIN {X 0.212,Y -565.413,Z 1218.955,A 0.000,B 0.000,C 90.000,E1 27.847} C_DIS
LIN {X 0.006,Y -561.309,Z 1218.951,A 0.000,B 0.000,C 90.000,E1 27.180} C_DIS
LIN {X 0.108,Y -557.835,Z 1218.948,A 0.000,B 0.000,C 90.000,E1 26.616} C_DIS
LIN {X 0.189,Y -554.137,Z 1218.945,A 0.000,B 0.000,C 90.000,E1 26.052} C_DIS
LIN {X -0.138,Y -551.198,Z 1218.943,A 0.000,B 0.000,C 90.000,E1 25.668} C_DIS
LIN {X 0.133,Y -546.980,Z 1218.939,A 0.000,B 0.000,C 90.000,E1 25.079} C_DIS
LIN {X 0.011,Y -541.355,Z 1218.936,A 0.000,B 0.000,C 90.000,E1 24.387} C_DIS
LIN {X -0.161,Y -535.341,Z 1218.932,A 0.000,B 0.000,C 90.000,E1 23.695} C_DIS
LIN {X 0.326,Y -525.137,Z 1218.925,A 0.000,B 0.000,C 90.000,E1 22.514} C_DIS
LIN {X 0.131,Y -519.790,Z 1218.922,A 0.000,B 0.000,C 90.000,E1 21.972} C_DIS
LIN {X -0.064,Y -510.616,Z 1218.917,A 0.000,B 0.000,C 90.000,E1 21.046} C_DIS
LIN {X 0.175,Y -500.932,Z 1218.912,A 0.000,B 0.000,C 90.000,E1 20.066} C_DIS
LIN {X 0.106,Y -492.294,Z 1218.907,A 0.000,B 0.000,C 90.000,E1 19.268} C_DIS
LIN {X -0.087,Y -482.124,Z 1218.902,A 0.000,B 0.000,C 90.000,E1 18.362} C_DIS
LIN {X -0.149,Y -475.068,Z 1218.899,A 0.000,B 0.000,C 90.000,E1 17.747} C_DIS
LIN {X 0.127,Y -457.544,Z 1218.890,A 0.000,B 0.000,C 90.000,E1 16.150} C_DIS
LIN {X -0.020,Y -441.333,Z 1218.881,A 0.000,B 0.000,C 90.000,E1 14.662} C_DIS
LIN {X 0.120,Y -421.143,Z 1218.870,A 0.000,B 0.000,C 90.000,E1 12.591} C_DIS
LIN {X -0.108,Y -403.008,Z 1218.859,A 0.000,B 0.000,C 90.000,E1 10.546} C_DIS
LIN {X -0.050,Y -397.758,Z 1218.855,A 0.000,B 0.000,C 90.000,E1 9.849} C_DIS
LIN {X 0.173,Y -395.003,Z 1218.852,A 0.000,B 0.000,C 90.000,E1 9.378} C_DIS
LIN {X 0.105,Y -394.337,Z 1218.851,A 0.000,B 0.000,C 90.000,E1 9.208} C_DIS
LIN {X 0.203,Y -393.650,Z 1218.850,A 0.000,B 0.000,C 90.000,E1 8.973} C_DIS
LIN {X 0.165,Y -393.639,Z 1218.850,A 0.000,B 0.000,C 90.000,E1 8.973} C_DIS
LIN {X 0.050,Y -393.844,Z 1218.849,A 0.000,B 0.000,C 90.000,E1 8.746} C_DIS
LIN {X 0.012,Y -393.856,Z 1218.849,A 0.000,B 0.000,C 90.000,E1 8.746} C_DIS
LIN {X 0.168,Y -396.863,Z 1218.845,A 0.000,B 0.000,C 90.000,E1 8.049} C_DIS
LIN {X 0.027,Y -400.354,Z 1218.843,A 0.000,B 0.000,C 90.000,E1 7.644} C_DIS
LIN {X 0.081,Y -403.882,Z 1218.841,A 0.000,B 0.000,C 90.000,E1 7.296} C_DIS
LIN {X 0.098,Y -407.262,Z 1218.839,A 0.000,B 0.000,C 90.000,E1 7.011} C_DIS
LIN {X -0.090,Y -421.291,Z 1218.833,A 0.000,B 0.000,C 90.000,E1 5.967} C_DIS
LIN {X -0.033,Y -432.483,Z 1218.828,A 0.000,B 0.000,C 90.000,E1 5.106} C_DIS
LIN {X 0.035,Y -443.607,Z 1218.824,A 0.000,B 0.000,C 90.000,E1 4.245} C_DIS
LIN {X 0.155,Y -456.297,Z 1218.818,A 0.000,B 0.000,C 90.000,E1 3.269} C_DIS
LIN {X -0.048,Y -466.983,Z 1218.814,A 0.000,B 0.000,C 90.000,E1 2.465} C_DIS
LIN {X 0.135,Y -473.061,Z 1218.811,A 0.000,B 0.000,C 90.000,E1 1.949} C_DIS
LIN {X 0.165,Y -479.031,Z 1218.808,A 0.000,B 0.000,C 90.000,E1 1.432} C_DIS
LIN {X 0.165,Y -484.716,Z 1218.805,A 0.000,B 0.000,C 90.000,E1 0.917} C_DIS
LIN {X 0.238,Y -491.607,Z 1218.802,A 0.000,B 0.000,C 90.000,E1 0.229} C_DIS
LIN {X 0.149,Y -498.603,Z 1218.797,A 0.000,B 0.000,C 90.000,E1 359.484} C_DIS
LIN {X 0.159,Y -504.962,Z 1218.793,A 0.000,B 0.000,C 90.000,E1 358.740} C_DIS
LIN {X -0.013,Y -509.743,Z 1218.790,A 0.000,B 0.000,C 90.000,E1 358.165} C_DIS
LIN {X 0.239,Y -516.188,Z 1218.785,A 0.000,B 0.000,C 90.000,E1 357.249} C_DIS
LIN {X 0.128,Y -520.230,Z 1218.782,A 0.000,B 0.000,C 90.000,E1 356.674} C_DIS
LIN {X -0.274,Y -524.880,Z 1218.778,A 0.000,B 0.000,C 90.000,E1 355.988} C_DIS
LIN {X 0.203,Y -528.337,Z 1218.774,A 0.000,B 0.000,C 90.000,E1 355.355} C_DIS
LIN {X -0.095,Y -532.208,Z 1218.770,A 0.000,B 0.000,C 90.000,E1 354.666} C_DIS
LIN {X -0.048,Y -536.350,Z 1218.766,A 0.000,B 0.000,C 90.000,E1 353.799} C_DIS
LIN {X 0.262,Y -538.311,Z 1218.763,A 0.000,B 0.000,C 90.000,E1 353.337} C_DIS
LIN {X -0.157,Y -542.992,Z 1218.757,A 0.000,B 0.000,C 90.000,E1 352.243} C_DIS
LIN {X 0.004,Y -546.049,Z 1218.752,A 0.000,B 0.000,C 90.000,E1 351.376} C_DIS
LIN {X 0.286,Y -548.828,Z 1218.747,A 0.000,B 0.000,C 90.000,E1 350.500} C_DIS
LIN {X -0.033,Y -551.316,Z 1218.743,A 0.000,B 0.000,C 90.000,E1 349.690} C_DIS
LIN {X -0.229,Y -553.661,Z 1218.738,A 0.000,B 0.000,C 90.000,E1 348.870} C_DIS
LIN {X 0.277,Y -556.559,Z 1218.732,A 0.000,B 0.000,C 90.000,E1 347.701} C_DIS
LIN {X -0.268,Y -559.153,Z 1218.726,A 0.000,B 0.000,C 90.000,E1 346.645} C_DIS
LIN {X 0.046,Y -562.069,Z 1218.718,A 0.000,B 0.000,C 90.000,E1 345.227} C_DIS
LIN {X 0.101,Y -563.694,Z 1218.713,A 0.000,B 0.000,C 90.000,E1 344.393} C_DIS
LIN {X -0.212,Y -565.740,Z 1218.707,A 0.000,B 0.000,C 90.000,E1 343.323} C_DIS
LIN {X 0.207,Y -567.508,Z 1218.701,A 0.000,B 0.000,C 90.000,E1 342.181} C_DIS
LIN {X -0.271,Y -569.472,Z 1218.694,A 0.000,B 0.000,C 90.000,E1 340.859} C_DIS
LIN {X 0.036,Y -570.455,Z 1218.689,A 0.000,B 0.000,C 90.000,E1 340.007} C_DIS
LIN {X -0.182,Y -571.232,Z 1218.684,A 0.000,B 0.000,C 90.000,E1 339.209} C_DIS
LIN {X 0.141,Y -571.799,Z 1218.680,A 0.000,B 0.000,C 90.000,E1 338.358} C_DIS
LIN {X -0.018,Y -572.022,Z 1218.674,A 0.000,B 0.000,C 90.000,E1 337.283} C_DIS
LIN {X -0.053,Y -571.971,Z 1218.671,A 0.000,B 0.000,C 90.000,E1 336.741} C_DIS
LIN {X 0.135,Y -571.803,Z 1218.668,A 0.000,B 0.000,C 90.000,E1 336.177} C_DIS
LIN {X 0.154,Y -571.179,Z 1218.663,A 0.000,B 0.000,C 90.000,E1 335.357} C_DIS
LIN {X -0.002,Y -569.838,Z 1218.657,A 0.000,B 0.000,C 90.000,E1 334.280} C_DIS
LIN {X -0.171,Y -569.488,Z 1218.656,A 0.000,B 0.000,C 90.000,E1 334.024} C_DIS
LIN {X -0.098,Y -567.270,Z 1218.650,A 0.000,B 0.000,C 90.000,E1 332.922} C_DIS
LIN {X 0.050,Y -566.012,Z 1218.646,A 0.000,B 0.000,C 90.000,E1 332.359} C_DIS
LIN {X 0.260,Y -563.796,Z 1218.642,A 0.000,B 0.000,C 90.000,E1 331.513} C_DIS
LIN {X -0.122,Y -561.903,Z 1218.639,A 0.000,B 0.000,C 90.000,E1 331.001} C_DIS
LIN {X -0.344,Y -559.104,Z 1218.635,A 0.000,B 0.000,C 90.000,E1 330.333} C_DIS
LIN {X 0.065,Y -555.018,Z 1218.630,A 0.000,B 0.000,C 90.000,E1 329.459} C_DIS
LIN {X 0.257,Y -551.143,Z 1218.627,A 0.000,B 0.000,C 90.000,E1 328.742} C_DIS
LIN {X 0.104,Y -545.699,Z 1218.622,A 0.000,B 0.000,C 90.000,E1 327.916} C_DIS
LIN {X -0.151,Y -543.843,Z 1218.620,A 0.000,B 0.000,C 90.000,E1 327.661} C_DIS
LIN {X 0.217,Y -538.489,Z 1218.616,A 0.000,B 0.000,C 90.000,E1 326.914} C_DIS
LIN {X 0.081,Y -530.635,Z 1218.611,A 0.000,B 0.000,C 90.000,E1 325.928} C_DIS
LIN {X 0.070,Y -519.056,Z 1218.603,A 0.000,B 0.000,C 90.000,E1 324.482} C_DIS
LIN {X -0.043,Y -515.023,Z 1218.599,A 0.000,B 0.000,C 90.000,E1 323.909} C_DIS
LIN {X -0.246,Y -512.066,Z 1218.597,A 0.000,B 0.000,C 90.000,E1 323.417} C_DIS
LIN {X -0.184,Y -510.252,Z 1218.594,A 0.000,B 0.000,C 90.000,E1 322.924} C_DIS
LIN {X 0.042,Y -509.519,Z 1218.592,A 0.000,B 0.000,C 90.000,E1 322.603} C_DIS
LIN {X -0.046,Y -508.957,Z 1218.591,A 0.000,B 0.000,C 90.000,E1 322.316} C_DIS
LIN {X 0.174,Y -508.388,Z 1218.587,A 0.000,B 0.000,C 90.000,E1 321.698} C_DIS
LIN {X 0.109,Y -508.175,Z 1218.581,A 0.000,B 0.000,C 90.000,E1 320.517} C_DIS
LIN {X 0.166,Y -509.668,Z 1218.566,A 0.000,B 0.000,C 90.000,E1 317.838} C_DIS
LIN {X 0.223,Y -510.672,Z 1218.556,A 0.000,B 0.000,C 90.000,E1 316.053} C_DIS
LIN {X 0.031,Y -511.460,Z 1218.548,A 0.000,B 0.000,C 90.000,E1 314.595} C_DIS
LIN {X 0.004,Y -512.384,Z 1218.536,A 0.000,B 0.000,C 90.000,E1 312.528} C_DIS
LIN {X -0.138,Y -513.133,Z 1218.528,A 0.000,B 0.000,C 90.000,E1 311.067} C_DIS
LIN {X 0.042,Y -513.938,Z 1218.518,A 0.000,B 0.000,C 90.000,E1 309.277} C_DIS
LIN {X 0.137,Y -514.253,Z 1218.513,A 0.000,B 0.000,C 90.000,E1 308.382} C_DIS
LIN {X 0.279,Y -515.074,Z 1218.500,A 0.000,B 0.000,C 90.000,E1 306.011} C_DIS
LIN {X -0.017,Y -515.795,Z 1218.490,A 0.000,B 0.000,C 90.000,E1 304.278} C_DIS
LIN {X 0.054,Y -516.307,Z 1218.482,A 0.000,B 0.000,C 90.000,E1 302.801} C_DIS
LIN {X -0.071,Y -516.767,Z 1218.473,A 0.000,B 0.000,C 90.000,E1 301.052} C_DIS
LIN {X 0.315,Y -516.924,Z 1218.468,A 0.000,B 0.000,C 90.000,E1 300.129} C_DIS
LIN {X -0.062,Y -517.119,Z 1218.458,A 0.000,B 0.000,C 90.000,E1 298.409} C_DIS
LIN {X 0.106,Y -517.259,Z 1218.450,A 0.000,B 0.000,C 90.000,E1 296.924} C_DIS
LIN {X -0.083,Y -517.302,Z 1218.443,A 0.000,B 0.000,C 90.000,E1 295.771} C_DIS
LIN {X -0.014,Y -517.392,Z 1218.433,A 0.000,B 0.000,C 90.000,E1 294.003} C_DIS
LIN {X 0.188,Y -517.449,Z 1218.425,A 0.000,B 0.000,C 90.000,E1 292.514} C_DIS
LIN {X 0.067,Y -517.395,Z 1218.419,A 0.000,B 0.000,C 90.000,E1 291.354} C_DIS
LIN {X 0.129,Y -516.951,Z 1218.412,A 0.000,B 0.000,C 90.000,E1 290.174} C_DIS
LIN {X 0.090,Y -516.169,Z 1218.402,A 0.000,B 0.000,C 90.000,E1 288.417} C_DIS
LIN {X -0.156,Y -515.205,Z 1218.391,A 0.000,B 0.000,C 90.000,E1 286.386} C_DIS
LIN {X 0.046,Y -513.736,Z 1218.378,A 0.000,B 0.000,C 90.000,E1 284.008} C_DIS
LIN {X 0.037,Y -512.856,Z 1218.370,A 0.000,B 0.000,C 90.000,E1 282.535} C_DIS
LIN {X -0.129,Y -511.641,Z 1218.360,A 0.000,B 0.000,C 90.000,E1 280.782} C_DIS
LIN {X 0.136,Y -510.284,Z 1218.348,A 0.000,B 0.000,C 90.000,E1 278.681} C_DIS
LIN {X -0.022,Y -508.649,Z 1218.333,A 0.000,B 0.000,C 90.000,E1 276.030} C_DIS
LIN {X 0.105,Y -507.783,Z 1218.325,A 0.000,B 0.000,C 90.000,E1 274.531} C_DIS
LIN {X 0.239,Y -507.152,Z 1218.319,A 0.000,B 0.000,C 90.000,E1 273.326} C_DIS
LIN {X -0.027,Y -505.651,Z 1218.305,A 0.000,B 0.000,C 90.000,E1 270.974} C_DIS
LIN {X 0.139,Y -504.245,Z 1218.292,A 0.000,B 0.000,C 90.000,E1 268.568} C_DIS
LIN {X -0.098,Y -503.022,Z 1218.281,A 0.000,B 0.000,C 90.000,E1 266.502} C_DIS
LIN {X -0.038,Y -502.244,Z 1218.274,A 0.000,B 0.000,C 90.000,E1 265.298} C_DIS
LIN {X -0.246,Y -500.588,Z 1218.262,A 0.000,B 0.000,C 90.000,E1 263.223} C_DIS
LIN {X -0.273,Y -499.247,Z 1218.254,A 0.000,B 0.000,C 90.000,E1 261.724} C_DIS
LIN {X 0.235,Y -497.638,Z 1218.244,A 0.000,B 0.000,C 90.000,E1 259.859} C_DIS
LIN {X 0.140,Y -495.848,Z 1218.232,A 0.000,B 0.000,C 90.000,E1 257.757} C_DIS
LIN {X 0.191,Y -494.513,Z 1218.222,A 0.000,B 0.000,C 90.000,E1 255.936} C_DIS
LIN {X -0.047,Y -493.406,Z 1218.214,A 0.000,B 0.000,C 90.000,E1 254.448} C_DIS
LIN {X 0.032,Y -491.800,Z 1218.197,A 0.000,B 0.000,C 90.000,E1 251.402} C_DIS
LIN {X 0.078,Y -490.967,Z 1218.187,A 0.000,B 0.000,C 90.000,E1 249.571} C_DIS
LIN {X 0.067,Y -490.016,Z 1218.178,A 0.000,B 0.000,C 90.000,E1 248.050} C_DIS
LIN {X -0.076,Y -489.101,Z 1218.171,A 0.000,B 0.000,C 90.000,E1 246.847} C_DIS
LIN {X 0.005,Y -488.357,Z 1218.166,A 0.000,B 0.000,C 90.000,E1 245.921} C_DIS
LIN {X -0.134,Y -486.922,Z 1218.158,A 0.000,B 0.000,C 90.000,E1 244.409} C_DIS
LIN {X -0.089,Y -485.366,Z 1218.149,A 0.000,B 0.000,C 90.000,E1 242.871} C_DIS
LIN {X -0.068,Y -484.337,Z 1218.144,A 0.000,B 0.000,C 90.000,E1 241.948} C_DIS
LIN {X -0.082,Y -482.505,Z 1218.136,A 0.000,B 0.000,C 90.000,E1 240.411} C_DIS
LIN {X 0.131,Y -480.340,Z 1218.125,A 0.000,B 0.000,C 90.000,E1 238.535} C_DIS
LIN {X -0.110,Y -478.841,Z 1218.118,A 0.000,B 0.000,C 90.000,E1 237.327} C_DIS
LIN {X 0.059,Y -476.345,Z 1218.106,A 0.000,B 0.000,C 90.000,E1 235.135} C_DIS
LIN {X -0.061,Y -473.945,Z 1218.094,A 0.000,B 0.000,C 90.000,E1 232.970} C_DIS
LIN {X -0.015,Y -471.057,Z 1218.079,A 0.000,B 0.000,C 90.000,E1 230.150} C_DIS
LIN {X 0.195,Y -469.351,Z 1218.068,A 0.000,B 0.000,C 90.000,E1 228.243} C_DIS
LIN {X 0.017,Y -467.576,Z 1218.058,A 0.000,B 0.000,C 90.000,E1 226.377} C_DIS
LIN {X -0.012,Y -465.305,Z 1218.042,A 0.000,B 0.000,C 90.000,E1 223.542} C_DIS
LIN {X 0.096,Y -464.939,Z 1218.000,A 0.000,B 0.000,C 90.000,E1 215.931} C_DIS
LIN {X 0.232,Y -466.505,Z 1217.982,A 0.000,B 0.000,C 90.000,E1 212.752} C_DIS
LIN {X -0.139,Y -468.512,Z 1217.970,A 0.000,B 0.000,C 90.000,E1 210.590} C_DIS
LIN {X -0.032,Y -471.945,Z 1217.952,A 0.000,B 0.000,C 90.000,E1 207.436} C_DIS
LIN {X 0.294,Y -474.621,Z 1217.940,A 0.000,B 0.000,C 90.000,E1 205.207} C_DIS
LIN {X -0.221,Y -481.929,Z 1217.914,A 0.000,B 0.000,C 90.000,E1 200.610} C_DIS
LIN {X -0.160,Y -489.003,Z 1217.896,A 0.000,B 0.000,C 90.000,E1 197.221} C_DIS
LIN {X -0.135,Y -496.603,Z 1217.879,A 0.000,B 0.000,C 90.000,E1 194.175} C_DIS
LIN {X -0.110,Y -502.507,Z 1217.867,A 0.000,B 0.000,C 90.000,E1 192.063} C_DIS
LIN {X 0.023,Y -507.527,Z 1217.857,A 0.000,B 0.000,C 90.000,E1 190.254} C_DIS
LIN {X 0.152,Y -513.732,Z 1217.845,A 0.000,B 0.000,C 90.000,E1 188.163} C_DIS
LIN {X -0.030,Y -517.335,Z 1217.839,A 0.000,B 0.000,C 90.000,E1 187.004} C_DIS
LIN {X -0.226,Y -520.856,Z 1217.832,A 0.000,B 0.000,C 90.000,E1 185.853} C_DIS
LIN {X 0.059,Y -526.039,Z 1217.823,A 0.000,B 0.000,C 90.000,E1 184.073} C_DIS
LIN {X -0.013,Y -529.531,Z 1217.816,A 0.000,B 0.000,C 90.000,E1 182.922} C_DIS
LIN {X -0.072,Y -533.000,Z 1217.810,A 0.000,B 0.000,C 90.000,E1 181.776} C_DIS
LIN {X -0.085,Y -538.179,Z 1217.800,A 0.000,B 0.000,C 90.000,E1 180.057} C_DIS
LIN {X -0.048,Y -540.716,Z 1217.796,A 0.000,B 0.000,C 90.000,E1 179.198} C_DIS
LIN {X 0.121,Y -545.715,Z 1217.786,A 0.000,B 0.000,C 90.000,E1 177.478} C_DIS
LIN {X -0.202,Y -549.685,Z 1217.778,A 0.000,B 0.000,C 90.000,E1 176.102} C_DIS
LIN {X 0.234,Y -554.295,Z 1217.769,A 0.000,B 0.000,C 90.000,E1 174.375} C_DIS
LIN {X 0.093,Y -557.995,Z 1217.761,A 0.000,B 0.000,C 90.000,E1 172.996} C_DIS
LIN {X 0.220,Y -562.326,Z 1217.752,A 0.000,B 0.000,C 90.000,E1 171.319} C_DIS
LIN {X -0.196,Y -565.931,Z 1217.744,A 0.000,B 0.000,C 90.000,E1 169.982} C_DIS
LIN {X 0.298,Y -570.148,Z 1217.735,A 0.000,B 0.000,C 90.000,E1 168.285} C_DIS
LIN {X 0.135,Y -573.737,Z 1217.728,A 0.000,B 0.000,C 90.000,E1 166.937} C_DIS
LIN {X 0.242,Y -579.694,Z 1217.715,A 0.000,B 0.000,C 90.000,E1 164.755} C_DIS
LIN {X -0.065,Y -586.731,Z 1217.702,A 0.000,B 0.000,C 90.000,E1 162.362} C_DIS
LIN {X -0.197,Y -596.279,Z 1217.686,A 0.000,B 0.000,C 90.000,E1 159.444} C_DIS
LIN {X -0.062,Y -602.087,Z 1217.677,A 0.000,B 0.000,C 90.000,E1 157.847} C_DIS
LIN {X -0.077,Y -606.962,Z 1217.670,A 0.000,B 0.000,C 90.000,E1 156.538} C_DIS
LIN {X -0.050,Y -612.622,Z 1217.661,A 0.000,B 0.000,C 90.000,E1 154.973} C_DIS
LIN {X -0.166,Y -616.348,Z 1217.655,A 0.000,B 0.000,C 90.000,E1 153.948} C_DIS
LIN {X 0.324,Y -619.863,Z 1217.650,A 0.000,B 0.000,C 90.000,E1 152.871} C_DIS
LIN {X -0.243,Y -624.937,Z 1217.641,A 0.000,B 0.000,C 90.000,E1 151.385} C_DIS
LIN {X 0.099,Y -628.281,Z 1217.635,A 0.000,B 0.000,C 90.000,E1 150.333} C_DIS
LIN {X 0.343,Y -633.884,Z 1217.625,A 0.000,B 0.000,C 90.000,E1 148.535} C_DIS
LIN {X -0.245,Y -637.713,Z 1217.618,A 0.000,B 0.000,C 90.000,E1 147.327} C_DIS
LIN {X -0.431,Y -641.297,Z 1217.611,A 0.000,B 0.000,C 90.000,E1 146.087} C_DIS
LIN {X -0.116,Y -643.311,Z 1217.607,A 0.000,B 0.000,C 90.000,E1 145.308} C_DIS
LIN {X 0.269,Y -645.854,Z 1217.602,A 0.000,B 0.000,C 90.000,E1 144.276} C_DIS
LIN {X 0.156,Y -648.163,Z 1217.596,A 0.000,B 0.000,C 90.000,E1 143.290} C_DIS
LIN {X 0.359,Y -652.102,Z 1217.587,A 0.000,B 0.000,C 90.000,E1 141.537} C_DIS
LIN {X 0.200,Y -655.298,Z 1217.578,A 0.000,B 0.000,C 90.000,E1 140.070} C_DIS
LIN {X 0.059,Y -657.949,Z 1217.572,A 0.000,B 0.000,C 90.000,E1 138.852} C_DIS
LIN {X -0.039,Y -660.673,Z 1217.565,A 0.000,B 0.000,C 90.000,E1 137.634} C_DIS
LIN {X 0.321,Y -664.890,Z 1217.554,A 0.000,B 0.000,C 90.000,E1 135.648} C_DIS
LIN {X 0.322,Y -669.521,Z 1217.543,A 0.000,B 0.000,C 90.000,E1 133.704} C_DIS
LIN {X -0.053,Y -673.789,Z 1217.534,A 0.000,B 0.000,C 90.000,E1 132.043} C_DIS
LIN {X -0.314,Y -677.356,Z 1217.526,A 0.000,B 0.000,C 90.000,E1 130.620} C_DIS
LIN {X 0.027,Y -680.950,Z 1217.518,A 0.000,B 0.000,C 90.000,E1 129.152} C_DIS
LIN {X -0.124,Y -683.932,Z 1217.511,A 0.000,B 0.000,C 90.000,E1 127.971} C_DIS
LIN {X 0.344,Y -687.515,Z 1217.503,A 0.000,B 0.000,C 90.000,E1 126.503} C_DIS
LIN {X 0.191,Y -689.268,Z 1217.499,A 0.000,B 0.000,C 90.000,E1 125.804} C_DIS
LIN {X -0.059,Y -692.534,Z 1217.491,A 0.000,B 0.000,C 90.000,E1 124.405} C_DIS
LIN {X 0.092,Y -695.148,Z 1217.485,A 0.000,B 0.000,C 90.000,E1 123.214} C_DIS
LIN {X -0.130,Y -697.230,Z 1217.479,A 0.000,B 0.000,C 90.000,E1 122.291} C_DIS
LIN {X -0.289,Y -699.581,Z 1217.473,A 0.000,B 0.000,C 90.000,E1 121.131} C_DIS
LIN {X 0.178,Y -701.827,Z 1217.466,A 0.000,B 0.000,C 90.000,E1 119.922} C_DIS
LIN {X 0.329,Y -703.897,Z 1217.460,A 0.000,B 0.000,C 90.000,E1 118.743} C_DIS
LIN {X -0.395,Y -704.950,Z 1217.456,A 0.000,B 0.000,C 90.000,E1 118.103} C_DIS
LIN {X -0.155,Y -705.723,Z 1217.452,A 0.000,B 0.000,C 90.000,E1 117.385} C_DIS
LIN {X 0.090,Y -706.211,Z 1217.448,A 0.000,B 0.000,C 90.000,E1 116.668} C_DIS
LIN {X 0.316,Y -706.625,Z 1217.443,A 0.000,B 0.000,C 90.000,E1 115.720} C_DIS
LIN {X 0.257,Y -706.493,Z 1217.439,A 0.000,B 0.000,C 90.000,E1 115.027} C_DIS
LIN {X -0.094,Y -706.189,Z 1217.437,A 0.000,B 0.000,C 90.000,E1 114.591} C_DIS
LIN {X -0.155,Y -705.339,Z 1217.434,A 0.000,B 0.000,C 90.000,E1 114.131} C_DIS
LIN {X -0.152,Y -704.811,Z 1217.433,A 0.000,B 0.000,C 90.000,E1 113.898} C_DIS
LIN {X 0.418,Y -702.691,Z 1217.430,A 0.000,B 0.000,C 90.000,E1 113.387} C_DIS
LIN {X -0.366,Y -702.104,Z 1217.430,A 0.000,B 0.000,C 90.000,E1 113.334} C_DIS
LIN {X -0.227,Y -701.245,Z 1217.429,A 0.000,B 0.000,C 90.000,E1 113.206} C_DIS
LIN {X -0.090,Y -699.973,Z 1217.428,A 0.000,B 0.000,C 90.000,E1 113.078} C_DIS
LIN {X 0.036,Y -694.504,Z 1217.426,A 0.000,B 0.000,C 90.000,E1 112.642} C_DIS
LIN {X 0.381,Y -692.409,Z 1217.425,A 0.000,B 0.000,C 90.000,E1 112.514} C_DIS
LIN {X 0.075,Y -685.864,Z 1217.424,A 0.000,B 0.000,C 90.000,E1 112.333} C_DIS
LIN {X -0.178,Y -684.489,Z 1217.424,A 0.000,B 0.000,C 90.000,E1 112.333} C_DIS
LIN {X 0.097,Y -677.514,Z 1217.424,A 0.000,B 0.000,C 90.000,E1 112.280} C_DIS
LIN {X 0.045,Y -612.450,Z 1217.424,A 0.000,B 0.000,C 90.000,E1 112.280} C_DIS
LIN {X -0.072,Y -610.753,Z 1217.423,A 0.000,B 0.000,C 90.000,E1 112.206} C_DIS
LIN {X 0.177,Y -606.545,Z 1217.422,A 0.000,B 0.000,C 90.000,E1 111.897} C_DIS
LIN {X -0.376,Y -605.125,Z 1217.421,A 0.000,B 0.000,C 90.000,E1 111.844} C_DIS
LIN {X -0.197,Y -602.617,Z 1217.420,A 0.000,B 0.000,C 90.000,E1 111.589} C_DIS
LIN {X 0.144,Y -601.774,Z 1217.419,A 0.000,B 0.000,C 90.000,E1 111.461} C_DIS
LIN {X 0.002,Y -600.111,Z 1217.418,A 0.000,B 0.000,C 90.000,E1 111.227} C_DIS
LIN {X -0.038,Y -599.745,Z 1217.417,A 0.000,B 0.000,C 90.000,E1 111.099} C_DIS
LIN {X -0.124,Y -600.183,Z 1217.416,A 0.000,B 0.000,C 90.000,E1 110.844} C_DIS
LIN {X 0.336,Y -601.645,Z 1217.413,A 0.000,B 0.000,C 90.000,E1 110.301} C_DIS
LIN {X -0.329,Y -604.534,Z 1217.409,A 0.000,B 0.000,C 90.000,E1 109.577} C_DIS
LIN {X -0.119,Y -606.266,Z 1217.406,A 0.000,B 0.000,C 90.000,E1 109.033} C_DIS
LIN {X 0.265,Y -613.008,Z 1217.394,A 0.000,B 0.000,C 90.000,E1 106.913} C_DIS
LIN {X 0.016,Y -613.721,Z 1217.393,A 0.000,B 0.000,C 90.000,E1 106.677} C_DIS
LIN {X 0.117,Y -615.583,Z 1217.390,A 0.000,B 0.000,C 90.000,E1 106.150} C_DIS
LIN {X -0.190,Y -617.168,Z 1217.387,A 0.000,B 0.000,C 90.000,E1 105.662} C_DIS
LIN {X -0.129,Y -619.118,Z 1217.383,A 0.000,B 0.000,C 90.000,E1 104.883} C_DIS
LIN {X 0.015,Y -620.190,Z 1217.380,A 0.000,B 0.000,C 90.000,E1 104.356} C_DIS
LIN {X -0.049,Y -621.364,Z 1217.375,A 0.000,B 0.000,C 90.000,E1 103.592} C_DIS
LIN {X 0.118,Y -621.818,Z 1217.373,A 0.000,B 0.000,C 90.000,E1 103.063} C_DIS
LIN {X 0.289,Y -621.838,Z 1217.370,A 0.000,B 0.000,C 90.000,E1 102.535} C_DIS
LIN {X -0.145,Y -621.525,Z 1217.367,A 0.000,B 0.000,C 90.000,E1 102.063} C_DIS
LIN {X 0.244,Y -621.279,Z 1217.366,A 0.000,B 0.000,C 90.000,E1 101.771} C_DIS
LIN {X -0.198,Y -620.449,Z 1217.363,A 0.000,B 0.000,C 90.000,E1 101.299} C_DIS
LIN {X -0.154,Y -619.196,Z 1217.360,A 0.000,B 0.000,C 90.000,E1 100.782} C_DIS
LIN {X -0.002,Y -617.670,Z 1217.357,A 0.000,B 0.000,C 90.000,E1 100.254} C_DIS
LIN {X -0.233,Y -616.699,Z 1217.356,A 0.000,B 0.000,C 90.000,E1 100.018} C_DIS
LIN {X -0.205,Y -614.294,Z 1217.353,A 0.000,B 0.000,C 90.000,E1 99.500} C_DIS
LIN {X -0.095,Y -611.670,Z 1217.350,A 0.000,B 0.000,C 90.000,E1 98.973} C_DIS
LIN {X -0.099,Y -608.356,Z 1217.347,A 0.000,B 0.000,C 90.000,E1 98.454} C_DIS
LIN {X -0.122,Y -604.272,Z 1217.344,A 0.000,B 0.000,C 90.000,E1 97.936} C_DIS
LIN {X -0.092,Y -599.548,Z 1217.341,A 0.000,B 0.000,C 90.000,E1 97.409} C_DIS
LIN {X -0.099,Y -592.926,Z 1217.338,A 0.000,B 0.000,C 90.000,E1 96.777} C_DIS
LIN {X -0.089,Y -585.608,Z 1217.334,A 0.000,B 0.000,C 90.000,E1 96.201} C_DIS
LIN {X -0.245,Y -579.117,Z 1217.332,A 0.000,B 0.000,C 90.000,E1 95.796} C_DIS
LIN {X -0.253,Y -573.868,Z 1217.331,A 0.000,B 0.000,C 90.000,E1 95.511} C_DIS
LIN {X 0.084,Y -572.270,Z 1217.330,A 0.000,B 0.000,C 90.000,E1 95.391} C_DIS
LIN {X 0.042,Y -567.740,Z 1217.328,A 0.000,B 0.000,C 90.000,E1 95.106} C_DIS
LIN {X -0.140,Y -564.397,Z 1217.326,A 0.000,B 0.000,C 90.000,E1 94.645} C_DIS
LIN {X 0.188,Y -563.895,Z 1217.324,A 0.000,B 0.000,C 90.000,E1 94.302} C_DIS
LIN {X -0.261,Y -563.953,Z 1217.319,A 0.000,B 0.000,C 90.000,E1 93.383} C_DIS
LIN {X -0.031,Y -565.185,Z 1217.308,A 0.000,B 0.000,C 90.000,E1 91.432} C_DIS
LIN {X 0.081,Y -566.371,Z 1217.299,A 0.000,B 0.000,C 90.000,E1 89.771} C_DIS
LIN {X -0.213,Y -567.789,Z 1217.288,A 0.000,B 0.000,C 90.000,E1 87.879} C_DIS
LIN {X 0.125,Y -569.219,Z 1217.277,A 0.000,B 0.000,C 90.000,E1 85.927} C_DIS
LIN {X 0.096,Y -571.049,Z 1217.265,A 0.000,B 0.000,C 90.000,E1 83.742} C_DIS
LIN {X -0.147,Y -572.479,Z 1217.256,A 0.000,B 0.000,C 90.000,E1 82.129} C_DIS
LIN {X 0.168,Y -573.553,Z 1217.249,A 0.000,B 0.000,C 90.000,E1 80.735} C_DIS
LIN {X -0.262,Y -574.355,Z 1217.243,A 0.000,B 0.000,C 90.000,E1 79.690} C_DIS
LIN {X -0.161,Y -575.373,Z 1217.234,A 0.000,B 0.000,C 90.000,E1 78.049} C_DIS
LIN {X -0.244,Y -576.184,Z 1217.226,A 0.000,B 0.000,C 90.000,E1 76.700} C_DIS
LIN {X 0.030,Y -577.060,Z 1217.217,A 0.000,B 0.000,C 90.000,E1 75.046} C_DIS
LIN {X -0.081,Y -577.904,Z 1217.208,A 0.000,B 0.000,C 90.000,E1 73.433} C_DIS
LIN {X 0.204,Y -578.981,Z 1217.197,A 0.000,B 0.000,C 90.000,E1 71.511} C_DIS
LIN {X -0.084,Y -579.766,Z 1217.190,A 0.000,B 0.000,C 90.000,E1 70.188} C_DIS
LIN {X 0.075,Y -581.069,Z 1217.179,A 0.000,B 0.000,C 90.000,E1 68.284} C_DIS
LIN {X -0.045,Y -582.641,Z 1217.169,A 0.000,B 0.000,C 90.000,E1 66.410} C_DIS
LIN {X 0.125,Y -583.935,Z 1217.161,A 0.000,B 0.000,C 90.000,E1 65.049} C_DIS
LIN {X 0.039,Y -585.622,Z 1217.151,A 0.000,B 0.000,C 90.000,E1 63.179} C_DIS
LIN {X 0.008,Y -587.549,Z 1217.141,A 0.000,B 0.000,C 90.000,E1 61.307} C_DIS
LIN {X -0.281,Y -588.947,Z 1217.133,A 0.000,B 0.000,C 90.000,E1 59.999} C_DIS
LIN {X -0.254,Y -590.209,Z 1217.126,A 0.000,B 0.000,C 90.000,E1 58.663} C_DIS
LIN {X -0.208,Y -591.440,Z 1217.118,A 0.000,B 0.000,C 90.000,E1 57.327} C_DIS
LIN {X 0.171,Y -592.514,Z 1217.111,A 0.000,B 0.000,C 90.000,E1 55.960} C_DIS
LIN {X 0.073,Y -593.587,Z 1217.104,A 0.000,B 0.000,C 90.000,E1 54.642} C_DIS
LIN {X 0.309,Y -595.010,Z 1217.093,A 0.000,B 0.000,C 90.000,E1 52.763} C_DIS
LIN {X 0.133,Y -595.958,Z 1217.086,A 0.000,B 0.000,C 90.000,E1 51.457} C_DIS
LIN {X -0.260,Y -596.659,Z 1217.080,A 0.000,B 0.000,C 90.000,E1 50.436} C_DIS
LIN {X -0.041,Y -597.224,Z 1217.073,A 0.000,B 0.000,C 90.000,E1 49.094} C_DIS
LIN {X 0.137,Y -597.772,Z 1217.065,A 0.000,B 0.000,C 90.000,E1 47.757} C_DIS
LIN {X -0.079,Y -598.135,Z 1217.058,A 0.000,B 0.000,C 90.000,E1 46.458} C_DIS
LIN {X 0.118,Y -598.313,Z 1217.054,A 0.000,B 0.000,C 90.000,E1 45.648} C_DIS
LIN {X 0.103,Y -598.256,Z 1217.048,A 0.000,B 0.000,C 90.000,E1 44.595} C_DIS
LIN {X 0.085,Y -598.045,Z 1217.042,A 0.000,B 0.000,C 90.000,E1 43.542} C_DIS
LIN {X -0.129,Y -597.382,Z 1217.035,A 0.000,B 0.000,C 90.000,E1 42.243} C_DIS
LIN {X 0.271,Y -596.855,Z 1217.029,A 0.000,B 0.000,C 90.000,E1 41.148} C_DIS
LIN {X 0.267,Y -596.167,Z 1217.023,A 0.000,B 0.000,C 90.000,E1 40.092} C_DIS
LIN {X -0.126,Y -595.391,Z 1217.017,A 0.000,B 0.000,C 90.000,E1 39.072} C_DIS
LIN {X -0.156,Y -594.456,Z 1217.011,A 0.000,B 0.000,C 90.000,E1 38.016} C_DIS
LIN {X -0.322,Y -593.591,Z 1217.007,A 0.000,B 0.000,C 90.000,E1 37.237} C_DIS
LIN {X 0.077,Y -592.234,Z 1217.001,A 0.000,B 0.000,C 90.000,E1 36.137} C_DIS
LIN {X -0.036,Y -590.071,Z 1216.993,A 0.000,B 0.000,C 90.000,E1 34.818} C_DIS
LIN {X -0.378,Y -587.824,Z 1216.988,A 0.000,B 0.000,C 90.000,E1 33.785} C_DIS
LIN {X 0.009,Y -586.601,Z 1216.985,A 0.000,B 0.000,C 90.000,E1 33.214} C_DIS
LIN {X 0.107,Y -583.548,Z 1216.979,A 0.000,B 0.000,C 90.000,E1 32.133} C_DIS
LIN {X 0.140,Y -581.935,Z 1216.976,A 0.000,B 0.000,C 90.000,E1 31.592} C_DIS
LIN {X 0.019,Y -578.980,Z 1216.971,A 0.000,B 0.000,C 90.000,E1 30.797} C_DIS
LIN {X 0.021,Y -576.815,Z 1216.968,A 0.000,B 0.000,C 90.000,E1 30.256} C_DIS
LIN {X -0.074,Y -573.858,Z 1216.964,A 0.000,B 0.000,C 90.000,E1 29.589} C_DIS
LIN {X 0.105,Y -571.220,Z 1216.961,A 0.000,B 0.000,C 90.000,E1 29.027} C_DIS
LIN {X 0.043,Y -568.411,Z 1216.958,A 0.000,B 0.000,C 90.000,E1 28.487} C_DIS
LIN {X 0.365,Y -564.587,Z 1216.955,A 0.000,B 0.000,C 90.000,E1 27.769} C_DIS
LIN {X -0.110,Y -560.433,Z 1216.951,A 0.000,B 0.000,C 90.000,E1 27.129} C_DIS
LIN {X 0.135,Y -556.054,Z 1216.947,A 0.000,B 0.000,C 90.000,E1 26.411} C_DIS
LIN {X 0.088,Y -551.219,Z 1216.943,A 0.000,B 0.000,C 90.000,E1 25.720} C_DIS
LIN {X 0.124,Y -547.064,Z 1216.940,A 0.000,B 0.000,C 90.000,E1 25.155} C_DIS
LIN {X 0.210,Y -542.652,Z 1216.937,A 0.000,B 0.000,C 90.000,E1 24.591} C_DIS
LIN {X 0.054,Y -536.755,Z 1216.933,A 0.000,B 0.000,C 90.000,E1 23.898} C_DIS
LIN {X -0.176,Y -529.238,Z 1216.928,A 0.000,B 0.000,C 90.000,E1 23.078} C_DIS
LIN {X 0.168,Y -522.756,Z 1216.924,A 0.000,B 0.000,C 90.000,E1 22.333} C_DIS
LIN {X -0.007,Y -513.584,Z 1216.919,A 0.000,B 0.000,C 90.000,E1 21.408} C_DIS
LIN {X -0.071,Y -506.884,Z 1216.915,A 0.000,B 0.000,C 90.000,E1 20.737} C_DIS
LIN {X -0.076,Y -500.007,Z 1216.911,A 0.000,B 0.000,C 90.000,E1 20.066} C_DIS
LIN {X -0.122,Y -491.374,Z 1216.907,A 0.000,B 0.000,C 90.000,E1 19.268} C_DIS
LIN {X -0.016,Y -482.984,Z 1216.903,A 0.000,B 0.000,C 90.000,E1 18.489} C_DIS
LIN {X -0.259,Y -474.458,Z 1216.899,A 0.000,B 0.000,C 90.000,E1 17.764} C_DIS
LIN {X 0.040,Y -458.597,Z 1216.891,A 0.000,B 0.000,C 90.000,E1 16.315} C_DIS
LIN {X -0.035,Y -438.157,Z 1216.880,A 0.000,B 0.000,C 90.000,E1 14.411} C_DIS
LIN {X 0.024,Y -421.035,Z 1216.870,A 0.000,B 0.000,C 90.000,E1 12.647} C_DIS
LIN {X -0.145,Y -404.483,Z 1216.860,A 0.000,B 0.000,C 90.000,E1 10.782} C_DIS
LIN {X 0.128,Y -397.988,Z 1216.855,A 0.000,B 0.000,C 90.000,E1 9.905} C_DIS
LIN {X 0.112,Y -395.754,Z 1216.853,A 0.000,B 0.000,C 90.000,E1 9.557} C_DIS
LIN {X 0.202,Y -394.530,Z 1216.852,A 0.000,B 0.000,C 90.000,E1 9.321} C_DIS
LIN {X -0.162,Y -393.610,Z 1216.850,A 0.000,B 0.000,C 90.000,E1 9.029} C_DIS
LIN {X 0.188,Y -393.609,Z 1216.850,A 0.000,B 0.000,C 90.000,E1 8.973} C_DIS
LIN {X 0.073,Y -393.839,Z 1216.849,A 0.000,B 0.000,C 90.000,E1 8.746} C_DIS
LIN {X 0.034,Y -393.845,Z 1216.849,A 0.000,B 0.000,C 90.000,E1 8.746} C_DIS
LIN {X 0.142,Y -396.611,Z 1216.845,A 0.000,B 0.000,C 90.000,E1 8.106} C_DIS
LIN {X -0.077,Y -397.126,Z 1216.845,A 0.000,B 0.000,C 90.000,E1 8.049} C_DIS
LIN {X -0.075,Y -401.462,Z 1216.842,A 0.000,B 0.000,C 90.000,E1 7.530} C_DIS
LIN {X -0.010,Y -405.196,Z 1216.840,A 0.000,B 0.000,C 90.000,E1 7.182} C_DIS
LIN {X -0.176,Y -424.180,Z 1216.832,A 0.000,B 0.000,C 90.000,E1 5.739} C_DIS
LIN {X -0.186,Y -438.484,Z 1216.826,A 0.000,B 0.000,C 90.000,E1 4.645} C_DIS
LIN {X -0.050,Y -452.557,Z 1216.820,A 0.000,B 0.000,C 90.000,E1 3.555} C_DIS
LIN {X 0.180,Y -461.980,Z 1216.816,A 0.000,B 0.000,C 90.000,E1 2.808} C_DIS
LIN {X -0.022,Y -468.178,Z 1216.813,A 0.000,B 0.000,C 90.000,E1 2.350} C_DIS
LIN {X 0.146,Y -474.248,Z 1216.810,A 0.000,B 0.000,C 90.000,E1 1.835} C_DIS
LIN {X -0.125,Y -478.707,Z 1216.808,A 0.000,B 0.000,C 90.000,E1 1.489} C_DIS
LIN {X -0.201,Y -484.527,Z 1216.805,A 0.000,B 0.000,C 90.000,E1 0.974} C_DIS
LIN {X 0.131,Y -491.219,Z 1216.802,A 0.000,B 0.000,C 90.000,E1 0.286} C_DIS
LIN {X -0.059,Y -497.398,Z 1216.798,A 0.000,B 0.000,C 90.000,E1 359.656} C_DIS
LIN {X 0.222,Y -505.032,Z 1216.793,A 0.000,B 0.000,C 90.000,E1 358.740} C_DIS
LIN {X -0.079,Y -510.835,Z 1216.789,A 0.000,B 0.000,C 90.000,E1 358.051} C_DIS
LIN {X -0.036,Y -516.228,Z 1216.785,A 0.000,B 0.000,C 90.000,E1 357.306} C_DIS
LIN {X -0.149,Y -520.318,Z 1216.782,A 0.000,B 0.000,C 90.000,E1 356.731} C_DIS
LIN {X -0.029,Y -524.988,Z 1216.778,A 0.000,B 0.000,C 90.000,E1 355.988} C_DIS
LIN {X -0.075,Y -528.485,Z 1216.775,A 0.000,B 0.000,C 90.000,E1 355.412} C_DIS
LIN {X 0.157,Y -532.372,Z 1216.771,A 0.000,B 0.000,C 90.000,E1 354.666} C_DIS
LIN {X -0.053,Y -535.890,Z 1216.766,A 0.000,B 0.000,C 90.000,E1 353.970} C_DIS
LIN {X -0.015,Y -538.525,Z 1216.763,A 0.000,B 0.000,C 90.000,E1 353.394} C_DIS
LIN {X 0.106,Y -543.237,Z 1216.757,A 0.000,B 0.000,C 90.000,E1 352.243} C_DIS
LIN {X -0.269,Y -546.316,Z 1216.752,A 0.000,B 0.000,C 90.000,E1 351.432} C_DIS
LIN {X 0.026,Y -549.977,Z 1216.746,A 0.000,B 0.000,C 90.000,E1 350.274} C_DIS
LIN {X 0.050,Y -553.940,Z 1216.738,A 0.000,B 0.000,C 90.000,E1 348.870} C_DIS
LIN {X 0.017,Y -556.842,Z 1216.732,A 0.000,B 0.000,C 90.000,E1 347.757} C_DIS
LIN {X 0.164,Y -560.068,Z 1216.724,A 0.000,B 0.000,C 90.000,E1 346.353} C_DIS
LIN {X -0.051,Y -562.943,Z 1216.717,A 0.000,B 0.000,C 90.000,E1 344.991} C_DIS
LIN {X -0.063,Y -565.577,Z 1216.709,A 0.000,B 0.000,C 90.000,E1 343.614} C_DIS
LIN {X 0.033,Y -567.051,Z 1216.704,A 0.000,B 0.000,C 90.000,E1 342.779} C_DIS
LIN {X 0.091,Y -569.126,Z 1216.697,A 0.000,B 0.000,C 90.000,E1 341.402} C_DIS
LIN {X -0.143,Y -570.252,Z 1216.692,A 0.000,B 0.000,C 90.000,E1 340.604} C_DIS
LIN {X -0.204,Y -571.479,Z 1216.686,A 0.000,B 0.000,C 90.000,E1 339.518} C_DIS
LIN {X 0.122,Y -572.143,Z 1216.682,A 0.000,B 0.000,C 90.000,E1 338.666} C_DIS
LIN {X -0.226,Y -572.460,Z 1216.679,A 0.000,B 0.000,C 90.000,E1 338.156} C_DIS
LIN {X -0.062,Y -572.640,Z 1216.672,A 0.000,B 0.000,C 90.000,E1 337.050} C_DIS
LIN {X -0.035,Y -572.465,Z 1216.668,A 0.000,B 0.000,C 90.000,E1 336.230} C_DIS
LIN {X -0.005,Y -571.936,Z 1216.663,A 0.000,B 0.000,C 90.000,E1 335.409} C_DIS
LIN {X 0.020,Y -571.008,Z 1216.659,A 0.000,B 0.000,C 90.000,E1 334.588} C_DIS
LIN {X 0.200,Y -570.306,Z 1216.656,A 0.000,B 0.000,C 90.000,E1 334.024} C_DIS
LIN {X -0.137,Y -569.295,Z 1216.653,A 0.000,B 0.000,C 90.000,E1 333.512} C_DIS
LIN {X 0.111,Y -567.533,Z 1216.648,A 0.000,B 0.000,C 90.000,E1 332.666} C_DIS
LIN {X 0.077,Y -565.490,Z 1216.644,A 0.000,B 0.000,C 90.000,E1 331.847} C_DIS
LIN {X 0.161,Y -564.738,Z 1216.642,A 0.000,B 0.000,C 90.000,E1 331.563} C_DIS
LIN {X -0.212,Y -562.948,Z 1216.639,A 0.000,B 0.000,C 90.000,E1 331.051} C_DIS
LIN {X 0.086,Y -561.943,Z 1216.638,A 0.000,B 0.000,C 90.000,E1 330.745} C_DIS
LIN {X -0.138,Y -559.032,Z 1216.634,A 0.000,B 0.000,C 90.000,E1 330.078} C_DIS
LIN {X -0.102,Y -555.574,Z 1216.630,A 0.000,B 0.000,C 90.000,E1 329.380} C_DIS
LIN {X 0.099,Y -551.629,Z 1216.626,A 0.000,B 0.000,C 90.000,E1 328.663} C_DIS
LIN {X -0.044,Y -546.164,Z 1216.621,A 0.000,B 0.000,C 90.000,E1 327.837} C_DIS
LIN {X 0.032,Y -543.168,Z 1216.619,A 0.000,B 0.000,C 90.000,E1 327.406} C_DIS
LIN {X 0.094,Y -536.672,Z 1216.614,A 0.000,B 0.000,C 90.000,E1 326.548} C_DIS
LIN {X -0.347,Y -530.949,Z 1216.610,A 0.000,B 0.000,C 90.000,E1 325.881} C_DIS
LIN {X 0.047,Y -519.405,Z 1216.602,A 0.000,B 0.000,C 90.000,E1 324.402} C_DIS
LIN {X -0.189,Y -515.742,Z 1216.599,A 0.000,B 0.000,C 90.000,E1 323.909} C_DIS
LIN {X 0.083,Y -512.737,Z 1216.597,A 0.000,B 0.000,C 90.000,E1 323.371} C_DIS
LIN {X -0.054,Y -510.251,Z 1216.593,A 0.000,B 0.000,C 90.000,E1 322.763} C_DIS
LIN {X 0.072,Y -509.307,Z 1216.590,A 0.000,B 0.000,C 90.000,E1 322.271} C_DIS
LIN {X -0.109,Y -508.710,Z 1216.587,A 0.000,B 0.000,C 90.000,E1 321.698} C_DIS
LIN {X -0.170,Y -508.493,Z 1216.581,A 0.000,B 0.000,C 90.000,E1 320.517} C_DIS
LIN {X 0.136,Y -509.591,Z 1216.569,A 0.000,B 0.000,C 90.000,E1 318.405} C_DIS
LIN {X 0.042,Y -510.294,Z 1216.563,A 0.000,B 0.000,C 90.000,E1 317.229} C_DIS
LIN {X 0.210,Y -511.178,Z 1216.554,A 0.000,B 0.000,C 90.000,E1 315.729} C_DIS
LIN {X 0.027,Y -511.931,Z 1216.546,A 0.000,B 0.000,C 90.000,E1 314.271} C_DIS
LIN {X -0.079,Y -513.084,Z 1216.533,A 0.000,B 0.000,C 90.000,E1 311.919} C_DIS
LIN {X -0.209,Y -513.796,Z 1216.525,A 0.000,B 0.000,C 90.000,E1 310.458} C_DIS
LIN {X 0.058,Y -514.508,Z 1216.516,A 0.000,B 0.000,C 90.000,E1 308.955} C_DIS
LIN {X -0.308,Y -514.934,Z 1216.508,A 0.000,B 0.000,C 90.000,E1 307.523} C_DIS
LIN {X 0.063,Y -515.525,Z 1216.500,A 0.000,B 0.000,C 90.000,E1 306.011} C_DIS
LIN {X 0.067,Y -516.279,Z 1216.490,A 0.000,B 0.000,C 90.000,E1 304.246} C_DIS
LIN {X 0.292,Y -516.801,Z 1216.482,A 0.000,B 0.000,C 90.000,E1 302.752} C_DIS
LIN {X 0.185,Y -517.306,Z 1216.472,A 0.000,B 0.000,C 90.000,E1 301.003} C_DIS
LIN {X 0.134,Y -517.443,Z 1216.468,A 0.000,B 0.000,C 90.000,E1 300.129} C_DIS
LIN {X 0.224,Y -517.660,Z 1216.458,A 0.000,B 0.000,C 90.000,E1 298.359} C_DIS
LIN {X 0.075,Y -517.849,Z 1216.448,A 0.000,B 0.000,C 90.000,E1 296.616} C_DIS
LIN {X -0.167,Y -517.908,Z 1216.437,A 0.000,B 0.000,C 90.000,E1 294.591} C_DIS
LIN {X -0.079,Y -518.005,Z 1216.427,A 0.000,B 0.000,C 90.000,E1 292.823} C_DIS
LIN {X -0.055,Y -517.970,Z 1216.419,A 0.000,B 0.000,C 90.000,E1 291.354} C_DIS
LIN {X 0.017,Y -517.524,Z 1216.412,A 0.000,B 0.000,C 90.000,E1 290.174} C_DIS
LIN {X -0.141,Y -516.921,Z 1216.404,A 0.000,B 0.000,C 90.000,E1 288.725} C_DIS
LIN {X -0.213,Y -515.915,Z 1216.393,A 0.000,B 0.000,C 90.000,E1 286.677} C_DIS
LIN {X -0.145,Y -515.379,Z 1216.388,A 0.000,B 0.000,C 90.000,E1 285.788} C_DIS
LIN {X -0.020,Y -514.301,Z 1216.378,A 0.000,B 0.000,C 90.000,E1 284.008} C_DIS
LIN {X -0.019,Y -513.416,Z 1216.370,A 0.000,B 0.000,C 90.000,E1 282.535} C_DIS
LIN {X -0.172,Y -512.199,Z 1216.360,A 0.000,B 0.000,C 90.000,E1 280.782} C_DIS
LIN {X 0.109,Y -510.908,Z 1216.348,A 0.000,B 0.000,C 90.000,E1 278.681} C_DIS
LIN {X -0.029,Y -509.265,Z 1216.333,A 0.000,B 0.000,C 90.000,E1 276.030} C_DIS
LIN {X 0.111,Y -508.401,Z 1216.325,A 0.000,B 0.000,C 90.000,E1 274.531} C_DIS
LIN {X -0.253,Y -507.749,Z 1216.319,A 0.000,B 0.000,C 90.000,E1 273.383} C_DIS
LIN {X 0.004,Y -506.282,Z 1216.305,A 0.000,B 0.000,C 90.000,E1 270.974} C_DIS
LIN {X 0.206,Y -505.719,Z 1216.301,A 0.000,B 0.000,C 90.000,E1 270.057} C_DIS
LIN {X 0.191,Y -504.913,Z 1216.292,A 0.000,B 0.000,C 90.000,E1 268.568} C_DIS
LIN {X -0.029,Y -503.666,Z 1216.281,A 0.000,B 0.000,C 90.000,E1 266.502} C_DIS
LIN {X 0.039,Y -502.878,Z 1216.274,A 0.000,B 0.000,C 90.000,E1 265.298} C_DIS
LIN {X -0.077,Y -501.491,Z 1216.264,A 0.000,B 0.000,C 90.000,E1 263.514} C_DIS
LIN {X -0.022,Y -500.132,Z 1216.256,A 0.000,B 0.000,C 90.000,E1 262.008} C_DIS
LIN {X 0.094,Y -498.999,Z 1216.249,A 0.000,B 0.000,C 90.000,E1 260.792} C_DIS
LIN {X 0.185,Y -497.953,Z 1216.242,A 0.000,B 0.000,C 90.000,E1 259.577} C_DIS
LIN {X 0.275,Y -496.500,Z 1216.232,A 0.000,B 0.000,C 90.000,E1 257.757} C_DIS
LIN {X -0.140,Y -495.132,Z 1216.222,A 0.000,B 0.000,C 90.000,E1 255.992} C_DIS
LIN {X 0.114,Y -494.076,Z 1216.214,A 0.000,B 0.000,C 90.000,E1 254.448} C_DIS
LIN {X 0.215,Y -492.390,Z 1216.197,A 0.000,B 0.000,C 90.000,E1 251.402} C_DIS
LIN {X 0.200,Y -491.816,Z 1216.190,A 0.000,B 0.000,C 90.000,E1 250.188} C_DIS
LIN {X -0.287,Y -491.142,Z 1216.183,A 0.000,B 0.000,C 90.000,E1 249.028} C_DIS
LIN {X -0.117,Y -490.109,Z 1216.175,A 0.000,B 0.000,C 90.000,E1 247.486} C_DIS
LIN {X 0.197,Y -489.144,Z 1216.168,A 0.000,B 0.000,C 90.000,E1 246.230} C_DIS
LIN {X 0.093,Y -487.387,Z 1216.158,A 0.000,B 0.000,C 90.000,E1 244.409} C_DIS
LIN {X 0.146,Y -485.809,Z 1216.149,A 0.000,B 0.000,C 90.000,E1 242.871} C_DIS
LIN {X 0.168,Y -484.314,Z 1216.143,A 0.000,B 0.000,C 90.000,E1 241.641} C_DIS
LIN {X -0.255,Y -482.893,Z 1216.136,A 0.000,B 0.000,C 90.000,E1 240.461} C_DIS
LIN {X -0.025,Y -480.699,Z 1216.125,A 0.000,B 0.000,C 90.000,E1 238.584} C_DIS
LIN {X 0.147,Y -479.167,Z 1216.119,A 0.000,B 0.000,C 90.000,E1 237.327} C_DIS
LIN {X 0.137,Y -477.054,Z 1216.108,A 0.000,B 0.000,C 90.000,E1 235.468} C_DIS
LIN {X 0.136,Y -474.579,Z 1216.096,A 0.000,B 0.000,C 90.000,E1 233.290} C_DIS
LIN {X 0.167,Y -473.576,Z 1216.091,A 0.000,B 0.000,C 90.000,E1 232.351} C_DIS
LIN {X 0.120,Y -470.758,Z 1216.075,A 0.000,B 0.000,C 90.000,E1 229.542} C_DIS
LIN {X -0.024,Y -468.987,Z 1216.065,A 0.000,B 0.000,C 90.000,E1 227.676} C_DIS
LIN {X -0.205,Y -467.195,Z 1216.054,A 0.000,B 0.000,C 90.000,E1 225.810} C_DIS
LIN {X 0.150,Y -465.889,Z 1216.046,A 0.000,B 0.000,C 90.000,E1 224.190} C_DIS
LIN {X -0.166,Y -464.110,Z 1216.019,A 0.000,B 0.000,C 90.000,E1 219.483} C_DIS
LIN {X -0.012,Y -464.771,Z 1216.002,A 0.000,B 0.000,C 90.000,E1 216.297} C_DIS
LIN {X -0.064,Y -465.452,Z 1215.991,A 0.000,B 0.000,C 90.000,E1 214.405} C_DIS
LIN {X -0.119,Y -466.358,Z 1215.982,A 0.000,B 0.000,C 90.000,E1 212.832} C_DIS
LIN {X -0.002,Y -468.063,Z 1215.972,A 0.000,B 0.000,C 90.000,E1 210.924} C_DIS
LIN {X -0.071,Y -471.027,Z 1215.956,A 0.000,B 0.000,C 90.000,E1 208.103} C_DIS
LIN {X -0.099,Y -472.878,Z 1215.947,A 0.000,B 0.000,C 90.000,E1 206.539} C_DIS
LIN {X 0.116,Y -474.846,Z 1215.939,A 0.000,B 0.000,C 90.000,E1 204.951} C_DIS
LIN {X 0.055,Y -482.318,Z 1215.913,A 0.000,B 0.000,C 90.000,E1 200.301} C_DIS
LIN {X 0.115,Y -488.842,Z 1215.896,A 0.000,B 0.000,C 90.000,E1 197.221} C_DIS
LIN {X 0.211,Y -494.846,Z 1215.882,A 0.000,B 0.000,C 90.000,E1 194.773} C_DIS
LIN {X -0.177,Y -500.676,Z 1215.870,A 0.000,B 0.000,C 90.000,E1 192.703} C_DIS
LIN {X 0.032,Y -504.141,Z 1215.864,A 0.000,B 0.000,C 90.000,E1 191.478} C_DIS
LIN {X -0.042,Y -512.828,Z 1215.847,A 0.000,B 0.000,C 90.000,E1 188.511} C_DIS
LIN {X 0.188,Y -517.387,Z 1215.839,A 0.000,B 0.000,C 90.000,E1 187.011} C_DIS
LIN {X 0.058,Y -520.971,Z 1215.833,A 0.000,B 0.000,C 90.000,E1 185.853} C_DIS
LIN {X -0.177,Y -526.178,Z 1215.823,A 0.000,B 0.000,C 90.000,E1 184.131} C_DIS
LIN {X -0.248,Y -529.696,Z 1215.816,A 0.000,B 0.000,C 90.000,E1 182.980} C_DIS
LIN {X 0.226,Y -533.192,Z 1215.810,A 0.000,B 0.000,C 90.000,E1 181.776} C_DIS
LIN {X 0.220,Y -538.427,Z 1215.801,A 0.000,B 0.000,C 90.000,E1 180.057} C_DIS
LIN {X 0.262,Y -540.985,Z 1215.796,A 0.000,B 0.000,C 90.000,E1 179.198} C_DIS
LIN {X -0.105,Y -546.040,Z 1215.786,A 0.000,B 0.000,C 90.000,E1 177.535} C_DIS
LIN {X 0.126,Y -550.063,Z 1215.778,A 0.000,B 0.000,C 90.000,E1 176.102} C_DIS
LIN {X 0.021,Y -554.715,Z 1215.769,A 0.000,B 0.000,C 90.000,E1 174.432} C_DIS
LIN {X -0.113,Y -558.482,Z 1215.761,A 0.000,B 0.000,C 90.000,E1 173.053} C_DIS
LIN {X 0.025,Y -562.899,Z 1215.752,A 0.000,B 0.000,C 90.000,E1 171.376} C_DIS
LIN {X 0.178,Y -566.576,Z 1215.745,A 0.000,B 0.000,C 90.000,E1 169.982} C_DIS
LIN {X 0.132,Y -570.880,Z 1215.735,A 0.000,B 0.000,C 90.000,E1 168.342} C_DIS
LIN {X -0.216,Y -573.802,Z 1215.729,A 0.000,B 0.000,C 90.000,E1 167.285} C_DIS
LIN {X 0.100,Y -579.039,Z 1215.719,A 0.000,B 0.000,C 90.000,E1 165.353} C_DIS
LIN {X -0.186,Y -582.891,Z 1215.711,A 0.000,B 0.000,C 90.000,E1 164.031} C_DIS
LIN {X 0.079,Y -588.498,Z 1215.701,A 0.000,B 0.000,C 90.000,E1 162.127} C_DIS
LIN {X 0.107,Y -597.207,Z 1215.686,A 0.000,B 0.000,C 90.000,E1 159.464} C_DIS
LIN {X -0.083,Y -602.927,Z 1215.677,A 0.000,B 0.000,C 90.000,E1 157.901} C_DIS
LIN {X -0.321,Y -607.702,Z 1215.670,A 0.000,B 0.000,C 90.000,E1 156.613} C_DIS
LIN {X 0.004,Y -612.377,Z 1215.663,A 0.000,B 0.000,C 90.000,E1 155.281} C_DIS
LIN {X 0.175,Y -616.051,Z 1215.657,A 0.000,B 0.000,C 90.000,E1 154.229} C_DIS
LIN {X 0.100,Y -619.559,Z 1215.651,A 0.000,B 0.000,C 90.000,E1 153.204} C_DIS
LIN {X 0.362,Y -623.717,Z 1215.644,A 0.000,B 0.000,C 90.000,E1 151.897} C_DIS
LIN {X 0.176,Y -628.664,Z 1215.636,A 0.000,B 0.000,C 90.000,E1 150.383} C_DIS
LIN {X 0.109,Y -634.191,Z 1215.626,A 0.000,B 0.000,C 90.000,E1 148.614} C_DIS
LIN {X -0.136,Y -637.943,Z 1215.619,A 0.000,B 0.000,C 90.000,E1 147.375} C_DIS
LIN {X -0.173,Y -640.793,Z 1215.613,A 0.000,B 0.000,C 90.000,E1 146.373} C_DIS
LIN {X 0.134,Y -642.804,Z 1215.609,A 0.000,B 0.000,C 90.000,E1 145.595} C_DIS
LIN {X 0.030,Y -645.963,Z 1215.602,A 0.000,B 0.000,C 90.000,E1 144.356} C_DIS
LIN {X 0.302,Y -648.228,Z 1215.597,A 0.000,B 0.000,C 90.000,E1 143.336} C_DIS
LIN {X 0.114,Y -652.123,Z 1215.587,A 0.000,B 0.000,C 90.000,E1 141.618} C_DIS
LIN {X -0.049,Y -655.297,Z 1215.579,A 0.000,B 0.000,C 90.000,E1 140.150} C_DIS
LIN {X -0.193,Y -657.936,Z 1215.572,A 0.000,B 0.000,C 90.000,E1 138.933} C_DIS
LIN {X -0.316,Y -661.163,Z 1215.564,A 0.000,B 0.000,C 90.000,E1 137.472} C_DIS
LIN {X 0.062,Y -664.840,Z 1215.554,A 0.000,B 0.000,C 90.000,E1 135.729} C_DIS
LIN {X 0.061,Y -669.411,Z 1215.543,A 0.000,B 0.000,C 90.000,E1 133.785} C_DIS
LIN {X 0.183,Y -673.666,Z 1215.534,A 0.000,B 0.000,C 90.000,E1 132.081} C_DIS
LIN {X -0.040,Y -677.803,Z 1215.525,A 0.000,B 0.000,C 90.000,E1 130.415} C_DIS
LIN {X -0.210,Y -681.409,Z 1215.517,A 0.000,B 0.000,C 90.000,E1 128.991} C_DIS
LIN {X 0.214,Y -684.964,Z 1215.509,A 0.000,B 0.000,C 90.000,E1 127.523} C_DIS
LIN {X 0.288,Y -688.588,Z 1215.501,A 0.000,B 0.000,C 90.000,E1 126.091} C_DIS
LIN {X -0.180,Y -691.294,Z 1215.494,A 0.000,B 0.000,C 90.000,E1 124.945} C_DIS
LIN {X -0.436,Y -693.991,Z 1215.488,A 0.000,B 0.000,C 90.000,E1 123.785} C_DIS
LIN {X 0.319,Y -696.661,Z 1215.481,A 0.000,B 0.000,C 90.000,E1 122.546} C_DIS
LIN {X 0.148,Y -699.035,Z 1215.474,A 0.000,B 0.000,C 90.000,E1 121.386} C_DIS
LIN {X -0.087,Y -701.741,Z 1215.467,A 0.000,B 0.000,C 90.000,E1 120.001} C_DIS
LIN {X -0.213,Y -703.418,Z 1215.462,A 0.000,B 0.000,C 90.000,E1 119.077} C_DIS
LIN {X 0.014,Y -704.540,Z 1215.458,A 0.000,B 0.000,C 90.000,E1 118.359} C_DIS
LIN {X -0.085,Y -705.737,Z 1215.452,A 0.000,B 0.000,C 90.000,E1 117.436} C_DIS
LIN {X -0.163,Y -706.232,Z 1215.449,A 0.000,B 0.000,C 90.000,E1 116.744} C_DIS
LIN {X 0.069,Y -706.650,Z 1215.443,A 0.000,B 0.000,C 90.000,E1 115.796} C_DIS
LIN {X 0.314,Y -706.558,Z 1215.440,A 0.000,B 0.000,C 90.000,E1 115.079} C_DIS
LIN {X -0.039,Y -706.279,Z 1215.437,A 0.000,B 0.000,C 90.000,E1 114.643} C_DIS
LIN {X 0.253,Y -705.971,Z 1215.436,A 0.000,B 0.000,C 90.000,E1 114.387} C_DIS
LIN {X -0.101,Y -705.086,Z 1215.433,A 0.000,B 0.000,C 90.000,E1 113.951} C_DIS
LIN {X 0.188,Y -702.991,Z 1215.430,A 0.000,B 0.000,C 90.000,E1 113.462} C_DIS
LIN {X -0.316,Y -702.443,Z 1215.430,A 0.000,B 0.000,C 90.000,E1 113.387} C_DIS
